	{attribute 'TcIecLibraryType'}
	{attribute 'external_name' := 'F_VN_FillContainerExp_DINT_GUID_B8D760C9_9A91_36E7_2F02_343FAF2948AF'}
	(* Partially fill the container with the specified value. Only possible for containers with basic elements. (expert function) *)
	FUNCTION F_VN_FillContainerExp_DINT : HRESULT
	VAR_INPUT
		ipContainer	:	ITcVnContainer;	(* Container with basic elements *)
		nValue	:	DINT;	(* Value to set the container elements *)
		nStartIdx	:	ULINT;	(* Start index *)
		nCount	:	ULINT;	(* Number of elements to set *)
		hrPrev	:	HRESULT;	(* HRESULT indicating the result of previous operations (If SUCCEEDED(hrPrev) equals false, no operation is executed.) *)
	END_VAR

END_FUNCTION

// Functions/Basic Container Operations/F_VN_FillContainerExp/F_VN_FillContainerExp_INT

	{attribute 'TcIecLibraryType'}
	{attribute 'external_name' := 'F_VN_FillContainerExp_INT_GUID_A3061951_E171_30F2_325A_8D22B4BE511B'}
	(* Partially fill the container with the specified value. Only possible for containers with basic elements. (expert function) *)
	FUNCTION F_VN_FillContainerExp_INT : HRESULT
	VAR_INPUT
		ipContainer	:	ITcVnContainer;	(* Container with basic elements *)
		nValue	:	INT;	(* Value to set the container elements *)
		nStartIdx	:	ULINT;	(* Start index *)
		nCount	:	ULINT;	(* Number of elements to set *)
		hrPrev	:	HRESULT;	(* HRESULT indicating the result of previous operations (If SUCCEEDED(hrPrev) equals false, no operation is executed.) *)
	END_VAR

END_FUNCTION

// Functions/Basic Container Operations/F_VN_FillContainerExp/F_VN_FillContainerExp_LREAL

	{attribute 'TcIecLibraryType'}
	{attribute 'external_name' := 'F_VN_FillContainerExp_LREAL_GUID_06A8F434_857D_380E_270C_C4307A69FA69'}
	(* Partially fill the container with the specified value. Only possible for containers with basic elements. (expert function) *)
	FUNCTION F_VN_FillContainerExp_LREAL : HRESULT
	VAR_INPUT
		ipContainer	:	ITcVnContainer;	(* Container with basic elements *)
		fValue	:	LREAL;	(* Value to set the container elements *)
		nStartIdx	:	ULINT;	(* Start index *)
		nCount	:	ULINT;	(* Number of elements to set *)
		hrPrev	:	HRESULT;	(* HRESULT indicating the result of previous operations (If SUCCEEDED(hrPrev) equals false, no operation is executed.) *)
	END_VAR

END_FUNCTION

// Functions/Basic Container Operations/F_VN_FillContainerExp/F_VN_FillContainerExp_REAL

	{attribute 'TcIecLibraryType'}
	{attribute 'external_name' := 'F_VN_FillContainerExp_REAL_GUID_48B84723_9FA9_3BC4_17C9_53CEC0ED83BA'}
	(* Partially fill the container with the specified value. Only possible for containers with basic elements. (expert function) *)
	FUNCTION F_VN_FillContainerExp_REAL : HRESULT
	VAR_INPUT
		ipContainer	:	ITcVnContainer;	(* Container with basic elements *)
		fValue	:	REAL;	(* Value to set the container elements *)
		nStartIdx	:	ULINT;	(* Start index *)
		nCount	:	ULINT;	(* Number of elements to set *)
		hrPrev	:	HRESULT;	(* HRESULT indicating the result of previous operations (If SUCCEEDED(hrPrev) equals false, no operation is executed.) *)
	END_VAR

END_FUNCTION

// Functions/Basic Container Operations/F_VN_FillContainerExp/F_VN_FillContainerExp_SINT

	{attribute 'TcIecLibraryType'}
	{attribute 'external_name' := 'F_VN_FillContainerExp_SINT_GUID_90863D28_18FF_36C8_1D3D_E4D2F13A07DE'}
	(* Partially fill the container with the specified value. Only possible for containers with basic elements. (expert function) *)
	FUNCTION F_VN_FillContainerExp_SINT : HRESULT
	VAR_INPUT
		ipContainer	:	ITcVnContainer;	(* Container with basic elements *)
		nValue	:	SINT;	(* Value to set the container elements *)
		nStartIdx	:	ULINT;	(* Start index *)
		nCount	:	ULINT;	(* Number of elements to set *)
		hrPrev	:	HRESULT;	(* HRESULT indicating the result of previous operations (If SUCCEEDED(hrPrev) equals false, no operation is executed.) *)
	END_VAR

END_FUNCTION

// Functions/Basic Container Operations/F_VN_FillContainerExp/F_VN_FillContainerExp_TcVnDMatch

	{attribute 'TcIecLibraryType'}
	{attribute 'external_name' := 'F_VN_FillContainerExp_TcVnDMatch_GUID_6EB328C8_9097_3649_0A18_3E606C0AB86C'}
	(* Partially fill the container with the specified value. Only possible for containers with basic elements. (expert function) *)
	FUNCTION F_VN_FillContainerExp_TcVnDMatch : HRESULT
	VAR_INPUT
		ipContainer	:	ITcVnContainer;	(* Container with basic elements *)
		stValue	:	REFERENCE TO TcVnDMatch;	(* Value to set the container elements *)
		nStartIdx	:	ULINT;	(* Start index *)
		nCount	:	ULINT;	(* Number of elements to set *)
		hrPrev	:	HRESULT;	(* HRESULT indicating the result of previous operations (If SUCCEEDED(hrPrev) equals false, no operation is executed.) *)
	END_VAR

END_FUNCTION

// Functions/Basic Container Operations/F_VN_FillContainerExp/F_VN_FillContainerExp_TcVnKeyPoint

	{attribute 'TcIecLibraryType'}
	{attribute 'external_name' := 'F_VN_FillContainerExp_TcVnKeyPoint_GUID_5E8CE577_86A2_3A7E_2E7B_5803657A1F81'}
	(* Partially fill the container with the specified value. Only possible for containers with basic elements. (expert function) *)
	FUNCTION F_VN_FillContainerExp_TcVnKeyPoint : HRESULT
	VAR_INPUT
		ipContainer	:	ITcVnContainer;	(* Container with basic elements *)
		stValue	:	REFERENCE TO TcVnKeyPoint;	(* Value to set the container elements *)
		nStartIdx	:	ULINT;	(* Start index *)
		nCount	:	ULINT;	(* Number of elements to set *)
		hrPrev	:	HRESULT;	(* HRESULT indicating the result of previous operations (If SUCCEEDED(hrPrev) equals false, no operation is executed.) *)
	END_VAR

END_FUNCTION

// Functions/Basic Container Operations/F_VN_FillContainerExp/F_VN_FillContainerExp_TcVnPoint2_DINT

	{attribute 'TcIecLibraryType'}
	{attribute 'external_name' := 'F_VN_FillContainerExp_TcVnPoint2_DINT_GUID_55F98272_BEB2_360C_30F1_C03770A26F61'}
	(* Partially fill the container with the specified value. Only possible for containers with basic elements. (expert function) *)
	FUNCTION F_VN_FillContainerExp_TcVnPoint2_DINT : HRESULT
	VAR_INPUT
		ipContainer	:	ITcVnContainer;	(* Container with basic elements *)
		aValue	:	REFERENCE TO TcVnPoint2_DINT;	(* Value to set the container elements *)
		nStartIdx	:	ULINT;	(* Start index *)
		nCount	:	ULINT;	(* Number of elements to set *)
		hrPrev	:	HRESULT;	(* HRESULT indicating the result of previous operations (If SUCCEEDED(hrPrev) equals false, no operation is executed.) *)
	END_VAR

END_FUNCTION

// Functions/Basic Container Operations/F_VN_FillContainerExp/F_VN_FillContainerExp_TcVnPoint2_LREAL

	{attribute 'TcIecLibraryType'}
	{attribute 'external_name' := 'F_VN_FillContainerExp_TcVnPoint2_LREAL_GUID_EFF1B11E_5960_30D8_0E25_714BE31C3872'}
	(* Partially fill the container with the specified value. Only possible for containers with basic elements. (expert function) *)
	FUNCTION F_VN_FillContainerExp_TcVnPoint2_LREAL : HRESULT
	VAR_INPUT
		ipContainer	:	ITcVnContainer;	(* Container with basic elements *)
		aValue	:	REFERENCE TO TcVnPoint2_LREAL;	(* Value to set the container elements *)
		nStartIdx	:	ULINT;	(* Start index *)
		nCount	:	ULINT;	(* Number of elements to set *)
		hrPrev	:	HRESULT;	(* HRESULT indicating the result of previous operations (If SUCCEEDED(hrPrev) equals false, no operation is executed.) *)
	END_VAR

END_FUNCTION

// Functions/Basic Container Operations/F_VN_FillContainerExp/F_VN_FillContainerExp_TcVnPoint2_REAL

	{attribute 'TcIecLibraryType'}
	{attribute 'external_name' := 'F_VN_FillContainerExp_TcVnPoint2_REAL_GUID_D2951393_83B9_352D_040D_B4C5DB5D1089'}
	(* Partially fill the container with the specified value. Only possible for containers with basic elements. (expert function) *)
	FUNCTION F_VN_FillContainerExp_TcVnPoint2_REAL : HRESULT
	VAR_INPUT
		ipContainer	:	ITcVnContainer;	(* Container with basic elements *)
		aValue	:	REFERENCE TO TcVnPoint2_REAL;	(* Value to set the container elements *)
		nStartIdx	:	ULINT;	(* Start index *)
		nCount	:	ULINT;	(* Number of elements to set *)
		hrPrev	:	HRESULT;	(* HRESULT indicating the result of previous operations (If SUCCEEDED(hrPrev) equals false, no operation is executed.) *)
	END_VAR

END_FUNCTION

// Functions/Basic Container Operations/F_VN_FillContainerExp/F_VN_FillContainerExp_TcVnPoint3_LREAL

	{attribute 'TcIecLibraryType'}
	{attribute 'external_name' := 'F_VN_FillContainerExp_TcVnPoint3_LREAL_GUID_B768B07E_F5CA_3309_10EA_C90BF763008C'}
	(* Partially fill the container with the specified value. Only possible for containers with basic elements. (expert function) *)
	FUNCTION F_VN_FillContainerExp_TcVnPoint3_LREAL : HRESULT
	VAR_INPUT
		ipContainer	:	ITcVnContainer;	(* Container with basic elements *)
		aValue	:	REFERENCE TO TcVnPoint3_LREAL;	(* Value to set the container elements *)
		nStartIdx	:	ULINT;	(* Start index *)
		nCount	:	ULINT;	(* Number of elements to set *)
		hrPrev	:	HRESULT;	(* HRESULT indicating the result of previous operations (If SUCCEEDED(hrPrev) equals false, no operation is executed.) *)
	END_VAR

END_FUNCTION

// Functions/Basic Container Operations/F_VN_FillContainerExp/F_VN_FillContainerExp_TcVnPoint3_REAL

	{attribute 'TcIecLibraryType'}
	{attribute 'external_name' := 'F_VN_FillContainerExp_TcVnPoint3_REAL_GUID_6AD4CB96_3415_3337_191D_E41E5C35A24A'}
	(* Partially fill the container with the specified value. Only possible for containers with basic elements. (expert function) *)
	FUNCTION F_VN_FillContainerExp_TcVnPoint3_REAL : HRESULT
	VAR_INPUT
		ipContainer	:	ITcVnContainer;	(* Container with basic elements *)
		aValue	:	REFERENCE TO TcVnPoint3_REAL;	(* Value to set the container elements *)
		nStartIdx	:	ULINT;	(* Start index *)
		nCount	:	ULINT;	(* Number of elements to set *)
		hrPrev	:	HRESULT;	(* HRESULT indicating the result of previous operations (If SUCCEEDED(hrPrev) equals false, no operation is executed.) *)
	END_VAR

END_FUNCTION

// Functions/Basic Container Operations/F_VN_FillContainerExp/F_VN_FillContainerExp_TcVnRectangle_DINT

	{attribute 'TcIecLibraryType'}
	{attribute 'external_name' := 'F_VN_FillContainerExp_TcVnRectangle_DINT_GUID_8BBC2A7F_64C7_3525_1E97_8C907D649B01'}
	(* Partially fill the container with the specified value. Only possible for containers with basic elements. (expert function) *)
	FUNCTION F_VN_FillContainerExp_TcVnRectangle_DINT : HRESULT
	VAR_INPUT
		ipContainer	:	ITcVnContainer;	(* Container with basic elements *)
		stValue	:	REFERENCE TO TcVnRectangle_DINT;	(* Value to set the container elements *)
		nStartIdx	:	ULINT;	(* Start index *)
		nCount	:	ULINT;	(* Number of elements to set *)
		hrPrev	:	HRESULT;	(* HRESULT indicating the result of previous operations (If SUCCEEDED(hrPrev) equals false, no operation is executed.) *)
	END_VAR

END_FUNCTION

// Functions/Basic Container Operations/F_VN_FillContainerExp/F_VN_FillContainerExp_TcVnVector2_DINT

	{attribute 'TcIecLibraryType'}
	{attribute 'external_name' := 'F_VN_FillContainerExp_TcVnVector2_DINT_GUID_D52E6A94_DE58_3796_0B33_2DB8E1E8C278'}
	(* Partially fill the container with the specified value. Only possible for containers with basic elements. (expert function) *)
	FUNCTION F_VN_FillContainerExp_TcVnVector2_DINT : HRESULT
	VAR_INPUT
		ipContainer	:	ITcVnContainer;	(* Container with basic elements *)
		aValue	:	REFERENCE TO TcVnVector2_DINT;	(* Value to set the container elements *)
		nStartIdx	:	ULINT;	(* Start index *)
		nCount	:	ULINT;	(* Number of elements to set *)
		hrPrev	:	HRESULT;	(* HRESULT indicating the result of previous operations (If SUCCEEDED(hrPrev) equals false, no operation is executed.) *)
	END_VAR

END_FUNCTION

// Functions/Basic Container Operations/F_VN_FillContainerExp/F_VN_FillContainerExp_TcVnVector2_INT

	{attribute 'TcIecLibraryType'}
	{attribute 'external_name' := 'F_VN_FillContainerExp_TcVnVector2_INT_GUID_F0AB717A_FE22_3EAE_3CD4_F3F145D668E6'}
	(* Partially fill the container with the specified value. Only possible for containers with basic elements. (expert function) *)
	FUNCTION F_VN_FillContainerExp_TcVnVector2_INT : HRESULT
	VAR_INPUT
		ipContainer	:	ITcVnContainer;	(* Container with basic elements *)
		aValue	:	REFERENCE TO TcVnVector2_INT;	(* Value to set the container elements *)
		nStartIdx	:	ULINT;	(* Start index *)
		nCount	:	ULINT;	(* Number of elements to set *)
		hrPrev	:	HRESULT;	(* HRESULT indicating the result of previous operations (If SUCCEEDED(hrPrev) equals false, no operation is executed.) *)
	END_VAR

END_FUNCTION

// Functions/Basic Container Operations/F_VN_FillContainerExp/F_VN_FillContainerExp_TcVnVector2_REAL

	{attribute 'TcIecLibraryType'}
	{attribute 'external_name' := 'F_VN_FillContainerExp_TcVnVector2_REAL_GUID_79D3ED73_D9A1_3766_3CCC_01A7C4952E54'}
	(* Partially fill the container with the specified value. Only possible for containers with basic elements. (expert function) *)
	FUNCTION F_VN_FillContainerExp_TcVnVector2_REAL : HRESULT
	VAR_INPUT
		ipContainer	:	ITcVnContainer;	(* Container with basic elements *)
		aValue	:	REFERENCE TO TcVnVector2_REAL;	(* Value to set the container elements *)
		nStartIdx	:	ULINT;	(* Start index *)
		nCount	:	ULINT;	(* Number of elements to set *)
		hrPrev	:	HRESULT;	(* HRESULT indicating the result of previous operations (If SUCCEEDED(hrPrev) equals false, no operation is executed.) *)
	END_VAR

END_FUNCTION

// Functions/Basic Container Operations/F_VN_FillContainerExp/F_VN_FillContainerExp_TcVnVector2_SINT

	{attribute 'TcIecLibraryType'}
	{attribute 'external_name' := 'F_VN_FillContainerExp_TcVnVector2_SINT_GUID_5A606FB7_F136_3298_1B9E_CE3509B64A28'}
	(* Partially fill the container with the specified value. Only possible for containers with basic elements. (expert function) *)
	FUNCTION F_VN_FillContainerExp_TcVnVector2_SINT : HRESULT
	VAR_INPUT
		ipContainer	:	ITcVnContainer;	(* Container with basic elements *)
		aValue	:	REFERENCE TO TcVnVector2_SINT;	(* Value to set the container elements *)
		nStartIdx	:	ULINT;	(* Start index *)
		nCount	:	ULINT;	(* Number of elements to set *)
		hrPrev	:	HRESULT;	(* HRESULT indicating the result of previous operations (If SUCCEEDED(hrPrev) equals false, no operation is executed.) *)
	END_VAR

END_FUNCTION

// Functions/Basic Container Operations/F_VN_FillContainerExp/F_VN_FillContainerExp_TcVnVector2_UINT

	{attribute 'TcIecLibraryType'}
	{attribute 'external_name' := 'F_VN_FillContainerExp_TcVnVector2_UINT_GUID_28D7E1DD_8953_3773_2801_6C09CC21C0E8'}
	(* Partially fill the container with the specified value. Only possible for containers with basic elements. (expert function) *)
	FUNCTION F_VN_FillContainerExp_TcVnVector2_UINT : HRESULT
	VAR_INPUT
		ipContainer	:	ITcVnContainer;	(* Container with basic elements *)
		aValue	:	REFERENCE TO TcVnVector2_UINT;	(* Value to set the container elements *)
		nStartIdx	:	ULINT;	(* Start index *)
		nCount	:	ULINT;	(* Number of elements to set *)
		hrPrev	:	HRESULT;	(* HRESULT indicating the result of previous operations (If SUCCEEDED(hrPrev) equals false, no operation is executed.) *)
	END_VAR

END_FUNCTION

// Functions/Basic Container Operations/F_VN_FillContainerExp/F_VN_FillContainerExp_TcVnVector2_USINT

	{attribute 'TcIecLibraryType'}
	{attribute 'external_name' := 'F_VN_FillContainerExp_TcVnVector2_USINT_GUID_CADE4DE9_E251_30AB_3613_56AF17179610'}
	(* Partially fill the container with the specified value. Only possible for containers with basic elements. (expert function) *)
	FUNCTION F_VN_FillContainerExp_TcVnVector2_USINT : HRESULT
	VAR_INPUT
		ipContainer	:	ITcVnContainer;	(* Container with basic elements *)
		aValue	:	REFERENCE TO TcVnVector2_USINT;	(* Value to set the container elements *)
		nStartIdx	:	ULINT;	(* Start index *)
		nCount	:	ULINT;	(* Number of elements to set *)
		hrPrev	:	HRESULT;	(* HRESULT indicating the result of previous operations (If SUCCEEDED(hrPrev) equals false, no operation is executed.) *)
	END_VAR

END_FUNCTION

// Functions/Basic Container Operations/F_VN_FillContainerExp/F_VN_FillContainerExp_TcVnVector3_INT

	{attribute 'TcIecLibraryType'}
	{attribute 'external_name' := 'F_VN_FillContainerExp_TcVnVector3_INT_GUID_8872692A_8B44_3770_16B3_D8C1614F2555'}
	(* Partially fill the container with the specified value. Only possible for containers with basic elements. (expert function) *)
	FUNCTION F_VN_FillContainerExp_TcVnVector3_INT : HRESULT
	VAR_INPUT
		ipContainer	:	ITcVnContainer;	(* Container with basic elements *)
		aValue	:	REFERENCE TO TcVnVector3_INT;	(* Value to set the container elements *)
		nStartIdx	:	ULINT;	(* Start index *)
		nCount	:	ULINT;	(* Number of elements to set *)
		hrPrev	:	HRESULT;	(* HRESULT indicating the result of previous operations (If SUCCEEDED(hrPrev) equals false, no operation is executed.) *)
	END_VAR

END_FUNCTION

// Functions/Basic Container Operations/F_VN_FillContainerExp/F_VN_FillContainerExp_TcVnVector3_REAL

	{attribute 'TcIecLibraryType'}
	{attribute 'external_name' := 'F_VN_FillContainerExp_TcVnVector3_REAL_GUID_F71E09F4_5F32_3920_383B_6FAF0F1CEF00'}
	(* Partially fill the container with the specified value. Only possible for containers with basic elements. (expert function) *)
	FUNCTION F_VN_FillContainerExp_TcVnVector3_REAL : HRESULT
	VAR_INPUT
		ipContainer	:	ITcVnContainer;	(* Container with basic elements *)
		aValue	:	REFERENCE TO TcVnVector3_REAL;	(* Value to set the container elements *)
		nStartIdx	:	ULINT;	(* Start index *)
		nCount	:	ULINT;	(* Number of elements to set *)
		hrPrev	:	HRESULT;	(* HRESULT indicating the result of previous operations (If SUCCEEDED(hrPrev) equals false, no operation is executed.) *)
	END_VAR

END_FUNCTION

// Functions/Basic Container Operations/F_VN_FillContainerExp/F_VN_FillContainerExp_TcVnVector3_SINT

	{attribute 'TcIecLibraryType'}
	{attribute 'external_name' := 'F_VN_FillContainerExp_TcVnVector3_SINT_GUID_C767BF5E_81CB_35B7_2F21_D703B6074D66'}
	(* Partially fill the container with the specified value. Only possible for containers with basic elements. (expert function) *)
	FUNCTION F_VN_FillContainerExp_TcVnVector3_SINT : HRESULT
	VAR_INPUT
		ipContainer	:	ITcVnContainer;	(* Container with basic elements *)
		aValue	:	REFERENCE TO TcVnVector3_SINT;	(* Value to set the container elements *)
		nStartIdx	:	ULINT;	(* Start index *)
		nCount	:	ULINT;	(* Number of elements to set *)
		hrPrev	:	HRESULT;	(* HRESULT indicating the result of previous operations (If SUCCEEDED(hrPrev) equals false, no operation is executed.) *)
	END_VAR

END_FUNCTION

// Functions/Basic Container Operations/F_VN_FillContainerExp/F_VN_FillContainerExp_TcVnVector3_UINT

	{attribute 'TcIecLibraryType'}
	{attribute 'external_name' := 'F_VN_FillContainerExp_TcVnVector3_UINT_GUID_A232C566_3D1F_3878_20BE_EC4C243376B7'}
	(* Partially fill the container with the specified value. Only possible for containers with basic elements. (expert function) *)
	FUNCTION F_VN_FillContainerExp_TcVnVector3_UINT : HRESULT
	VAR_INPUT
		ipContainer	:	ITcVnContainer;	(* Container with basic elements *)
		aValue	:	REFERENCE TO TcVnVector3_UINT;	(* Value to set the container elements *)
		nStartIdx	:	ULINT;	(* Start index *)
		nCount	:	ULINT;	(* Number of elements to set *)
		hrPrev	:	HRESULT;	(* HRESULT indicating the result of previous operations (If SUCCEEDED(hrPrev) equals false, no operation is executed.) *)
	END_VAR

END_FUNCTION

// Functions/Basic Container Operations/F_VN_FillContainerExp/F_VN_FillContainerExp_TcVnVector3_USINT

	{attribute 'TcIecLibraryType'}
	{attribute 'external_name' := 'F_VN_FillContainerExp_TcVnVector3_USINT_GUID_AF77E3C4_6637_32BB_0907_3628D17ABB88'}
	(* Partially fill the container with the specified value. Only possible for containers with basic elements. (expert function) *)
	FUNCTION F_VN_FillContainerExp_TcVnVector3_USINT : HRESULT
	VAR_INPUT
		ipContainer	:	ITcVnContainer;	(* Container with basic elements *)
		aValue	:	REFERENCE TO TcVnVector3_USINT;	(* Value to set the container elements *)
		nStartIdx	:	ULINT;	(* Start index *)
		nCount	:	ULINT;	(* Number of elements to set *)
		hrPrev	:	HRESULT;	(* HRESULT indicating the result of previous operations (If SUCCEEDED(hrPrev) equals false, no operation is executed.) *)
	END_VAR

END_FUNCTION

// Functions/Basic Container Operations/F_VN_FillContainerExp/F_VN_FillContainerExp_TcVnVector4_DINT

	{attribute 'TcIecLibraryType'}
	{attribute 'external_name' := 'F_VN_FillContainerExp_TcVnVector4_DINT_GUID_D0B471BF_D0B3_3250_3545_D00683C80B71'}
	(* Partially fill the container with the specified value. Only possible for containers with basic elements. (expert function) *)
	FUNCTION F_VN_FillContainerExp_TcVnVector4_DINT : HRESULT
	VAR_INPUT
		ipContainer	:	ITcVnContainer;	(* Container with basic elements *)
		aValue	:	REFERENCE TO TcVnVector4_DINT;	(* Value to set the container elements *)
		nStartIdx	:	ULINT;	(* Start index *)
		nCount	:	ULINT;	(* Number of elements to set *)
		hrPrev	:	HRESULT;	(* HRESULT indicating the result of previous operations (If SUCCEEDED(hrPrev) equals false, no operation is executed.) *)
	END_VAR

END_FUNCTION

// Functions/Basic Container Operations/F_VN_FillContainerExp/F_VN_FillContainerExp_TcVnVector4_INT

	{attribute 'TcIecLibraryType'}
	{attribute 'external_name' := 'F_VN_FillContainerExp_TcVnVector4_INT_GUID_FE07D4F2_2BAB_357F_1E6D_1BC89319641C'}
	(* Partially fill the container with the specified value. Only possible for containers with basic elements. (expert function) *)
	FUNCTION F_VN_FillContainerExp_TcVnVector4_INT : HRESULT
	VAR_INPUT
		ipContainer	:	ITcVnContainer;	(* Container with basic elements *)
		aValue	:	REFERENCE TO TcVnVector4_INT;	(* Value to set the container elements *)
		nStartIdx	:	ULINT;	(* Start index *)
		nCount	:	ULINT;	(* Number of elements to set *)
		hrPrev	:	HRESULT;	(* HRESULT indicating the result of previous operations (If SUCCEEDED(hrPrev) equals false, no operation is executed.) *)
	END_VAR

END_FUNCTION

// Functions/Basic Container Operations/F_VN_FillContainerExp/F_VN_FillContainerExp_TcVnVector4_LREAL

	{attribute 'TcIecLibraryType'}
	{attribute 'external_name' := 'F_VN_FillContainerExp_TcVnVector4_LREAL_GUID_DE917028_E855_3AAC_2584_39BC076C3EA3'}
	(* Partially fill the container with the specified value. Only possible for containers with basic elements. (expert function) *)
	FUNCTION F_VN_FillContainerExp_TcVnVector4_LREAL : HRESULT
	VAR_INPUT
		ipContainer	:	ITcVnContainer;	(* Container with basic elements *)
		aValue	:	REFERENCE TO TcVnVector4_LREAL;	(* Value to set the container elements *)
		nStartIdx	:	ULINT;	(* Start index *)
		nCount	:	ULINT;	(* Number of elements to set *)
		hrPrev	:	HRESULT;	(* HRESULT indicating the result of previous operations (If SUCCEEDED(hrPrev) equals false, no operation is executed.) *)
	END_VAR

END_FUNCTION

// Functions/Basic Container Operations/F_VN_FillContainerExp/F_VN_FillContainerExp_TcVnVector4_SINT

	{attribute 'TcIecLibraryType'}
	{attribute 'external_name' := 'F_VN_FillContainerExp_TcVnVector4_SINT_GUID_36AF45DF_9EEE_3748_11FA_C0473793B250'}
	(* Partially fill the container with the specified value. Only possible for containers with basic elements. (expert function) *)
	FUNCTION F_VN_FillContainerExp_TcVnVector4_SINT : HRESULT
	VAR_INPUT
		ipContainer	:	ITcVnContainer;	(* Container with basic elements *)
		aValue	:	REFERENCE TO TcVnVector4_SINT;	(* Value to set the container elements *)
		nStartIdx	:	ULINT;	(* Start index *)
		nCount	:	ULINT;	(* Number of elements to set *)
		hrPrev	:	HRESULT;	(* HRESULT indicating the result of previous operations (If SUCCEEDED(hrPrev) equals false, no operation is executed.) *)
	END_VAR

END_FUNCTION

// Functions/Basic Container Operations/F_VN_FillContainerExp/F_VN_FillContainerExp_TcVnVector4_UINT

	{attribute 'TcIecLibraryType'}
	{attribute 'external_name' := 'F_VN_FillContainerExp_TcVnVector4_UINT_GUID_6F025B14_1449_32FD_3652_7705ACD933FC'}
	(* Partially fill the container with the specified value. Only possible for containers with basic elements. (expert function) *)
	FUNCTION F_VN_FillContainerExp_TcVnVector4_UINT : HRESULT
	VAR_INPUT
		ipContainer	:	ITcVnContainer;	(* Container with basic elements *)
		aValue	:	REFERENCE TO TcVnVector4_UINT;	(* Value to set the container elements *)
		nStartIdx	:	ULINT;	(* Start index *)
		nCount	:	ULINT;	(* Number of elements to set *)
		hrPrev	:	HRESULT;	(* HRESULT indicating the result of previous operations (If SUCCEEDED(hrPrev) equals false, no operation is executed.) *)
	END_VAR

END_FUNCTION

// Functions/Basic Container Operations/F_VN_FillContainerExp/F_VN_FillContainerExp_TcVnVector4_USINT

	{attribute 'TcIecLibraryType'}
	{attribute 'external_name' := 'F_VN_FillContainerExp_TcVnVector4_USINT_GUID_88F61DD9_1D3A_3F92_2879_A4E50CB6EE10'}
	(* Partially fill the container with the specified value. Only possible for containers with basic elements. (expert function) *)
	FUNCTION F_VN_FillContainerExp_TcVnVector4_USINT : HRESULT
	VAR_INPUT
		ipContainer	:	ITcVnContainer;	(* Container with basic elements *)
		aValue	:	REFERENCE TO TcVnVector4_USINT;	(* Value to set the container elements *)
		nStartIdx	:	ULINT;	(* Start index *)
		nCount	:	ULINT;	(* Number of elements to set *)
		hrPrev	:	HRESULT;	(* HRESULT indicating the result of previous operations (If SUCCEEDED(hrPrev) equals false, no operation is executed.) *)
	END_VAR

END_FUNCTION

// Functions/Basic Container Operations/F_VN_FillContainerExp/F_VN_FillContainerExp_UDINT

	{attribute 'TcIecLibraryType'}
	{attribute 'external_name' := 'F_VN_FillContainerExp_UDINT_GUID_C1899B3C_8E1E_3688_3F00_9FEF7C4BAF80'}
	(* Partially fill the container with the specified value. Only possible for containers with basic elements. (expert function) *)
	FUNCTION F_VN_FillContainerExp_UDINT : HRESULT
	VAR_INPUT
		ipContainer	:	ITcVnContainer;	(* Container with basic elements *)
		nValue	:	UDINT;	(* Value to set the container elements *)
		nStartIdx	:	ULINT;	(* Start index *)
		nCount	:	ULINT;	(* Number of elements to set *)
		hrPrev	:	HRESULT;	(* HRESULT indicating the result of previous operations (If SUCCEEDED(hrPrev) equals false, no operation is executed.) *)
	END_VAR

END_FUNCTION

// Functions/Basic Container Operations/F_VN_FillContainerExp/F_VN_FillContainerExp_UINT

	{attribute 'TcIecLibraryType'}
	{attribute 'external_name' := 'F_VN_FillContainerExp_UINT_GUID_4625D03C_9DE0_3ACB_0D71_512E8D91ACEF'}
	(* Partially fill the container with the specified value. Only possible for containers with basic elements. (expert function) *)
	FUNCTION F_VN_FillContainerExp_UINT : HRESULT
	VAR_INPUT
		ipContainer	:	ITcVnContainer;	(* Container with basic elements *)
		nValue	:	UINT;	(* Value to set the container elements *)
		nStartIdx	:	ULINT;	(* Start index *)
		nCount	:	ULINT;	(* Number of elements to set *)
		hrPrev	:	HRESULT;	(* HRESULT indicating the result of previous operations (If SUCCEEDED(hrPrev) equals false, no operation is executed.) *)
	END_VAR

END_FUNCTION

// Functions/Basic Container Operations/F_VN_FillContainerExp/F_VN_FillContainerExp_ULINT

	{attribute 'TcIecLibraryType'}
	{attribute 'external_name' := 'F_VN_FillContainerExp_ULINT_GUID_E1571213_CE5E_37DB_3EDB_D35295DEA11A'}
	(* Partially fill the container with the specified value. Only possible for containers with basic elements. (expert function) *)
	FUNCTION F_VN_FillContainerExp_ULINT : HRESULT
	VAR_INPUT
		ipContainer	:	ITcVnContainer;	(* Container with basic elements *)
		nValue	:	ULINT;	(* Value to set the container elements *)
		nStartIdx	:	ULINT;	(* Start index *)
		nCount	:	ULINT;	(* Number of elements to set *)
		hrPrev	:	HRESULT;	(* HRESULT indicating the result of previous operations (If SUCCEEDED(hrPrev) equals false, no operation is executed.) *)
	END_VAR

END_FUNCTION

// Functions/Basic Container Operations/F_VN_FillContainerExp/F_VN_FillContainerExp_USINT

	{attribute 'TcIecLibraryType'}
	{attribute 'external_name' := 'F_VN_FillContainerExp_USINT_GUID_5EEE187D_276D_381A_26F0_6B86E27B5CD0'}
	(* Partially fill the container with the specified value. Only possible for containers with basic elements. (expert function) *)
	FUNCTION F_VN_FillContainerExp_USINT : HRESULT
	VAR_INPUT
		ipContainer	:	ITcVnContainer;	(* Container with basic elements *)
		nValue	:	USINT;	(* Value to set the container elements *)
		nStartIdx	:	ULINT;	(* Start index *)
		nCount	:	ULINT;	(* Number of elements to set *)
		hrPrev	:	HRESULT;	(* HRESULT indicating the result of previous operations (If SUCCEEDED(hrPrev) equals false, no operation is executed.) *)
	END_VAR

END_FUNCTION

// Functions/Basic Container Operations/F_VN_GetAt/F_VN_GetAt_ITcVnContainer

	{attribute 'TcIecLibraryType'}
	{attribute 'external_name' := 'F_VN_GetAt_ITcVnContainer_GUID_045FB529_DC44_35D8_25B4_376FBA31652E'}
	(* Gets the ITcVnContainer element at the specified index of the source container. (Alternatively use interface method .GetAt.) *)
	FUNCTION F_VN_GetAt_ITcVnContainer : HRESULT
	VAR_INPUT
		ipSrcContainer	:	ITcVnContainer;	(* Container with ITcVnContainer elements *)
		ipDestContainer	:	REFERENCE TO ITcVnContainer;	(* Returns the container at the specified index *)
		nIndex	:	ULINT;	(* Index of the requested element *)
		hrPrev	:	HRESULT;	(* HRESULT indicating the result of previous operations (If SUCCEEDED(hrPrev) equals false, no operation is executed.) *)
	END_VAR

END_FUNCTION

// Functions/Basic Container Operations/F_VN_GetAt/F_VN_GetAt_DINT

	{attribute 'TcIecLibraryType'}
	{attribute 'external_name' := 'F_VN_GetAt_DINT_GUID_D3F93AB3_14EE_32CD_0E8F_11068B05A3A3'}
	(* Gets the DINT element at the specified index of the container. *)
	FUNCTION F_VN_GetAt_DINT : HRESULT
	VAR_INPUT
		ipContainer	:	ITcVnContainer;	(* Container with DINT elements *)
		nElement	:	REFERENCE TO DINT;	(* Returns the element at the specified index *)
		nIndex	:	ULINT;	(* Index of the requested element *)
		hrPrev	:	HRESULT;	(* HRESULT indicating the result of previous operations (If SUCCEEDED(hrPrev) equals false, no operation is executed.) *)
	END_VAR

END_FUNCTION

// Functions/Basic Container Operations/F_VN_GetAt/F_VN_GetAt_INT

	{attribute 'TcIecLibraryType'}
	{attribute 'external_name' := 'F_VN_GetAt_INT_GUID_9B8341DD_2E11_3864_2634_BD22319F2AE6'}
	(* Gets the INT element at the specified index of the container. *)
	FUNCTION F_VN_GetAt_INT : HRESULT
	VAR_INPUT
		ipContainer	:	ITcVnContainer;	(* Container with INT elements *)
		nElement	:	REFERENCE TO INT;	(* Returns the element at the specified index *)
		nIndex	:	ULINT;	(* Index of the requested element *)
		hrPrev	:	HRESULT;	(* HRESULT indicating the result of previous operations (If SUCCEEDED(hrPrev) equals false, no operation is executed.) *)
	END_VAR

END_FUNCTION

// Functions/Basic Container Operations/F_VN_GetAt/F_VN_GetAt_LREAL

	{attribute 'TcIecLibraryType'}
	{attribute 'external_name' := 'F_VN_GetAt_LREAL_GUID_DC876A81_A8A4_3799_1F06_D74BAE2F1D06'}
	(* Gets the LREAL element at the specified index of the container. *)
	FUNCTION F_VN_GetAt_LREAL : HRESULT
	VAR_INPUT
		ipContainer	:	ITcVnContainer;	(* Container with LREAL elements *)
		fElement	:	REFERENCE TO LREAL;	(* Returns the element at the specified index *)
		nIndex	:	ULINT;	(* Index of the requested element *)
		hrPrev	:	HRESULT;	(* HRESULT indicating the result of previous operations (If SUCCEEDED(hrPrev) equals false, no operation is executed.) *)
	END_VAR

END_FUNCTION

// Functions/Basic Container Operations/F_VN_GetAt/F_VN_GetAt_REAL

	{attribute 'TcIecLibraryType'}
	{attribute 'external_name' := 'F_VN_GetAt_REAL_GUID_1E16943C_FBCF_3296_0945_06B3CBBED3E4'}
	(* Gets the REAL element at the specified index of the container. *)
	FUNCTION F_VN_GetAt_REAL : HRESULT
	VAR_INPUT
		ipContainer	:	ITcVnContainer;	(* Container with REAL elements *)
		fElement	:	REFERENCE TO REAL;	(* Returns the element at the specified index *)
		nIndex	:	ULINT;	(* Index of the requested element *)
		hrPrev	:	HRESULT;	(* HRESULT indicating the result of previous operations (If SUCCEEDED(hrPrev) equals false, no operation is executed.) *)
	END_VAR

END_FUNCTION

// Functions/Basic Container Operations/F_VN_GetAt/F_VN_GetAt_SINT

	{attribute 'TcIecLibraryType'}
	{attribute 'external_name' := 'F_VN_GetAt_SINT_GUID_881646F0_463E_317B_2E29_F707EE20003C'}
	(* Gets the SINT element at the specified index of the container. *)
	FUNCTION F_VN_GetAt_SINT : HRESULT
	VAR_INPUT
		ipContainer	:	ITcVnContainer;	(* Container with SINT elements *)
		nElement	:	REFERENCE TO SINT;	(* Returns the element at the specified index *)
		nIndex	:	ULINT;	(* Index of the requested element *)
		hrPrev	:	HRESULT;	(* HRESULT indicating the result of previous operations (If SUCCEEDED(hrPrev) equals false, no operation is executed.) *)
	END_VAR

END_FUNCTION

// Functions/Basic Container Operations/F_VN_GetAt/F_VN_GetAt_TcVnDMatch

	{attribute 'TcIecLibraryType'}
	{attribute 'external_name' := 'F_VN_GetAt_TcVnDMatch_GUID_3207E963_392F_3409_08E6_68F01287B943'}
	(* Gets the TcVnDMatch element at the specified index of the container. *)
	FUNCTION F_VN_GetAt_TcVnDMatch : HRESULT
	VAR_INPUT
		ipContainer	:	ITcVnContainer;	(* Container with TcVnDMatch elements *)
		stElement	:	REFERENCE TO TcVnDMatch;	(* Returns the element at the specified index *)
		nIndex	:	ULINT;	(* Index of the requested element *)
		hrPrev	:	HRESULT;	(* HRESULT indicating the result of previous operations (If SUCCEEDED(hrPrev) equals false, no operation is executed.) *)
	END_VAR

END_FUNCTION

// Functions/Basic Container Operations/F_VN_GetAt/F_VN_GetAt_TcVnKeyPoint

	{attribute 'TcIecLibraryType'}
	{attribute 'external_name' := 'F_VN_GetAt_TcVnKeyPoint_GUID_2D05125E_4551_301B_1496_C775451626E2'}
	(* Gets the TcVnKeyPoint element at the specified index of the container. *)
	FUNCTION F_VN_GetAt_TcVnKeyPoint : HRESULT
	VAR_INPUT
		ipContainer	:	ITcVnContainer;	(* Container with TcVnKeyPoint elements *)
		stElement	:	REFERENCE TO TcVnKeyPoint;	(* Returns the element at the specified index *)
		nIndex	:	ULINT;	(* Index of the requested element *)
		hrPrev	:	HRESULT;	(* HRESULT indicating the result of previous operations (If SUCCEEDED(hrPrev) equals false, no operation is executed.) *)
	END_VAR

END_FUNCTION

// Functions/Basic Container Operations/F_VN_GetAt/F_VN_GetAt_TcVnPoint2_DINT

	{attribute 'TcIecLibraryType'}
	{attribute 'external_name' := 'F_VN_GetAt_TcVnPoint2_DINT_GUID_E33E2091_0EF8_3437_0DF4_98D7E3EF7746'}
	(* Gets the TcVnPoint2_DINT element at the specified index of the container. *)
	FUNCTION F_VN_GetAt_TcVnPoint2_DINT : HRESULT
	VAR_INPUT
		ipContainer	:	ITcVnContainer;	(* Container with TcVnPoint2_DINT elements *)
		aElement	:	REFERENCE TO TcVnPoint2_DINT;	(* Returns the element at the specified index *)
		nIndex	:	ULINT;	(* Index of the requested element *)
		hrPrev	:	HRESULT;	(* HRESULT indicating the result of previous operations (If SUCCEEDED(hrPrev) equals false, no operation is executed.) *)
	END_VAR

END_FUNCTION

// Functions/Basic Container Operations/F_VN_GetAt/F_VN_GetAt_TcVnPoint2_LREAL

	{attribute 'TcIecLibraryType'}
	{attribute 'external_name' := 'F_VN_GetAt_TcVnPoint2_LREAL_GUID_9EEB5F99_0D0C_312C_2F99_C7BA67AF2141'}
	(* Gets the TcVnPoint2_LREAL element at the specified index of the container. *)
	FUNCTION F_VN_GetAt_TcVnPoint2_LREAL : HRESULT
	VAR_INPUT
		ipContainer	:	ITcVnContainer;	(* Container with TcVnPoint2_LREAL elements *)
		aElement	:	REFERENCE TO TcVnPoint2_LREAL;	(* Returns the element at the specified index *)
		nIndex	:	ULINT;	(* Index of the requested element *)
		hrPrev	:	HRESULT;	(* HRESULT indicating the result of previous operations (If SUCCEEDED(hrPrev) equals false, no operation is executed.) *)
	END_VAR

END_FUNCTION

// Functions/Basic Container Operations/F_VN_GetAt/F_VN_GetAt_TcVnPoint2_REAL

	{attribute 'TcIecLibraryType'}
	{attribute 'external_name' := 'F_VN_GetAt_TcVnPoint2_REAL_GUID_371EAF1D_26B5_3B9D_372A_6247762CF125'}
	(* Gets the TcVnPoint2_REAL element at the specified index of the container. *)
	FUNCTION F_VN_GetAt_TcVnPoint2_REAL : HRESULT
	VAR_INPUT
		ipContainer	:	ITcVnContainer;	(* Container with TcVnPoint2_REAL elements *)
		aElement	:	REFERENCE TO TcVnPoint2_REAL;	(* Returns the element at the specified index *)
		nIndex	:	ULINT;	(* Index of the requested element *)
		hrPrev	:	HRESULT;	(* HRESULT indicating the result of previous operations (If SUCCEEDED(hrPrev) equals false, no operation is executed.) *)
	END_VAR

END_FUNCTION

// Functions/Basic Container Operations/F_VN_GetAt/F_VN_GetAt_TcVnPoint3_LREAL

	{attribute 'TcIecLibraryType'}
	{attribute 'external_name' := 'F_VN_GetAt_TcVnPoint3_LREAL_GUID_90390C07_74BB_3F31_196C_51E52FA0FEDF'}
	(* Gets the TcVnPoint3_LREAL element at the specified index of the container. *)
	FUNCTION F_VN_GetAt_TcVnPoint3_LREAL : HRESULT
	VAR_INPUT
		ipContainer	:	ITcVnContainer;	(* Container with TcVnPoint3_LREAL elements *)
		aElement	:	REFERENCE TO TcVnPoint3_LREAL;	(* Returns the element at the specified index *)
		nIndex	:	ULINT;	(* Index of the requested element *)
		hrPrev	:	HRESULT;	(* HRESULT indicating the result of previous operations (If SUCCEEDED(hrPrev) equals false, no operation is executed.) *)
	END_VAR

END_FUNCTION

// Functions/Basic Container Operations/F_VN_GetAt/F_VN_GetAt_TcVnPoint3_REAL

	{attribute 'TcIecLibraryType'}
	{attribute 'external_name' := 'F_VN_GetAt_TcVnPoint3_REAL_GUID_0A5DCE69_37A2_35F9_0DF3_FEC0A8403AF7'}
	(* Gets the TcVnPoint3_REAL element at the specified index of the container. *)
	FUNCTION F_VN_GetAt_TcVnPoint3_REAL : HRESULT
	VAR_INPUT
		ipContainer	:	ITcVnContainer;	(* Container with TcVnPoint3_REAL elements *)
		aElement	:	REFERENCE TO TcVnPoint3_REAL;	(* Returns the element at the specified index *)
		nIndex	:	ULINT;	(* Index of the requested element *)
		hrPrev	:	HRESULT;	(* HRESULT indicating the result of previous operations (If SUCCEEDED(hrPrev) equals false, no operation is executed.) *)
	END_VAR

END_FUNCTION

// Functions/Basic Container Operations/F_VN_GetAt/F_VN_GetAt_TcVnRectangle_DINT

	{attribute 'TcIecLibraryType'}
	{attribute 'external_name' := 'F_VN_GetAt_TcVnRectangle_DINT_GUID_75B34143_A1C0_32FF_0BAA_7C7E335D62E6'}
	(* Gets the TcVnRectangle_DINT element at the specified index of the container. *)
	FUNCTION F_VN_GetAt_TcVnRectangle_DINT : HRESULT
	VAR_INPUT
		ipContainer	:	ITcVnContainer;	(* Container with TcVnRectangle_DINT elements *)
		stElement	:	REFERENCE TO TcVnRectangle_DINT;	(* Returns the element at the specified index *)
		nIndex	:	ULINT;	(* Index of the requested element *)
		hrPrev	:	HRESULT;	(* HRESULT indicating the result of previous operations (If SUCCEEDED(hrPrev) equals false, no operation is executed.) *)
	END_VAR

END_FUNCTION

// Functions/Basic Container Operations/F_VN_GetAt/F_VN_GetAt_TcVnVector2_DINT

	{attribute 'TcIecLibraryType'}
	{attribute 'external_name' := 'F_VN_GetAt_TcVnVector2_DINT_GUID_E7C2B37B_70C4_3998_2382_4EB9E1DE7BCE'}
	(* Gets the TcVnVector2_DINT element at the specified index of the container. *)
	FUNCTION F_VN_GetAt_TcVnVector2_DINT : HRESULT
	VAR_INPUT
		ipContainer	:	ITcVnContainer;	(* Container with TcVnVector2_DINT elements *)
		aElement	:	REFERENCE TO TcVnVector2_DINT;	(* Returns the element at the specified index *)
		nIndex	:	ULINT;	(* Index of the requested element *)
		hrPrev	:	HRESULT;	(* HRESULT indicating the result of previous operations (If SUCCEEDED(hrPrev) equals false, no operation is executed.) *)
	END_VAR

END_FUNCTION

// Functions/Basic Container Operations/F_VN_GetAt/F_VN_GetAt_TcVnVector2_INT

	{attribute 'TcIecLibraryType'}
	{attribute 'external_name' := 'F_VN_GetAt_TcVnVector2_INT_GUID_70115FDC_19E9_3A1A_170B_469E5110F923'}
	(* Gets the TcVnVector2_INT element at the specified index of the container. *)
	FUNCTION F_VN_GetAt_TcVnVector2_INT : HRESULT
	VAR_INPUT
		ipContainer	:	ITcVnContainer;	(* Container with TcVnVector2_INT elements *)
		aElement	:	REFERENCE TO TcVnVector2_INT;	(* Returns the element at the specified index *)
		nIndex	:	ULINT;	(* Index of the requested element *)
		hrPrev	:	HRESULT;	(* HRESULT indicating the result of previous operations (If SUCCEEDED(hrPrev) equals false, no operation is executed.) *)
	END_VAR

END_FUNCTION

// Functions/Basic Container Operations/F_VN_GetAt/F_VN_GetAt_TcVnVector2_REAL

	{attribute 'TcIecLibraryType'}
	{attribute 'external_name' := 'F_VN_GetAt_TcVnVector2_REAL_GUID_934F0AF6_F9AB_31D8_2BAB_3B9DF8D54B4F'}
	(* Gets the TcVnVector2_REAL element at the specified index of the container. *)
	FUNCTION F_VN_GetAt_TcVnVector2_REAL : HRESULT
	VAR_INPUT
		ipContainer	:	ITcVnContainer;	(* Container with TcVnVector2_REAL elements *)
		aElement	:	REFERENCE TO TcVnVector2_REAL;	(* Returns the element at the specified index *)
		nIndex	:	ULINT;	(* Index of the requested element *)
		hrPrev	:	HRESULT;	(* HRESULT indicating the result of previous operations (If SUCCEEDED(hrPrev) equals false, no operation is executed.) *)
	END_VAR

END_FUNCTION

// Functions/Basic Container Operations/F_VN_GetAt/F_VN_GetAt_TcVnVector2_SINT

	{attribute 'TcIecLibraryType'}
	{attribute 'external_name' := 'F_VN_GetAt_TcVnVector2_SINT_GUID_A03F3DE8_F80B_3551_2585_744B19853183'}
	(* Gets the TcVnVector2_SINT element at the specified index of the container. *)
	FUNCTION F_VN_GetAt_TcVnVector2_SINT : HRESULT
	VAR_INPUT
		ipContainer	:	ITcVnContainer;	(* Container with TcVnVector2_SINT elements *)
		aElement	:	REFERENCE TO TcVnVector2_SINT;	(* Returns the element at the specified index *)
		nIndex	:	ULINT;	(* Index of the requested element *)
		hrPrev	:	HRESULT;	(* HRESULT indicating the result of previous operations (If SUCCEEDED(hrPrev) equals false, no operation is executed.) *)
	END_VAR

END_FUNCTION

// Functions/Basic Container Operations/F_VN_GetAt/F_VN_GetAt_TcVnVector2_UINT

	{attribute 'TcIecLibraryType'}
	{attribute 'external_name' := 'F_VN_GetAt_TcVnVector2_UINT_GUID_C1EC9D9A_FD3C_3A6B_078C_FD8ED4C33F35'}
	(* Gets the TcVnVector2_UINT element at the specified index of the container. *)
	FUNCTION F_VN_GetAt_TcVnVector2_UINT : HRESULT
	VAR_INPUT
		ipContainer	:	ITcVnContainer;	(* Container with TcVnVector2_UINT elements *)
		aElement	:	REFERENCE TO TcVnVector2_UINT;	(* Returns the element at the specified index *)
		nIndex	:	ULINT;	(* Index of the requested element *)
		hrPrev	:	HRESULT;	(* HRESULT indicating the result of previous operations (If SUCCEEDED(hrPrev) equals false, no operation is executed.) *)
	END_VAR

END_FUNCTION

// Functions/Basic Container Operations/F_VN_GetAt/F_VN_GetAt_TcVnVector2_USINT

	{attribute 'TcIecLibraryType'}
	{attribute 'external_name' := 'F_VN_GetAt_TcVnVector2_USINT_GUID_9151A628_DCD5_3225_06FF_C1BAF6F1DAB4'}
	(* Gets the TcVnVector2_USINT element at the specified index of the container. *)
	FUNCTION F_VN_GetAt_TcVnVector2_USINT : HRESULT
	VAR_INPUT
		ipContainer	:	ITcVnContainer;	(* Container with TcVnVector2_USINT elements *)
		aElement	:	REFERENCE TO TcVnVector2_USINT;	(* Returns the element at the specified index *)
		nIndex	:	ULINT;	(* Index of the requested element *)
		hrPrev	:	HRESULT;	(* HRESULT indicating the result of previous operations (If SUCCEEDED(hrPrev) equals false, no operation is executed.) *)
	END_VAR

END_FUNCTION

// Functions/Basic Container Operations/F_VN_GetAt/F_VN_GetAt_TcVnVector3_INT

	{attribute 'TcIecLibraryType'}
	{attribute 'external_name' := 'F_VN_GetAt_TcVnVector3_INT_GUID_5314E713_0BA0_360B_1F6E_965C93ECA65C'}
	(* Gets the TcVnVector3_INT element at the specified index of the container. *)
	FUNCTION F_VN_GetAt_TcVnVector3_INT : HRESULT
	VAR_INPUT
		ipContainer	:	ITcVnContainer;	(* Container with TcVnVector3_INT elements *)
		aElement	:	REFERENCE TO TcVnVector3_INT;	(* Returns the element at the specified index *)
		nIndex	:	ULINT;	(* Index of the requested element *)
		hrPrev	:	HRESULT;	(* HRESULT indicating the result of previous operations (If SUCCEEDED(hrPrev) equals false, no operation is executed.) *)
	END_VAR

END_FUNCTION

// Functions/Basic Container Operations/F_VN_GetAt/F_VN_GetAt_TcVnVector3_REAL

	{attribute 'TcIecLibraryType'}
	{attribute 'external_name' := 'F_VN_GetAt_TcVnVector3_REAL_GUID_EF583C7F_272D_3493_1464_1CEFBDA69B47'}
	(* Gets the TcVnVector3_REAL element at the specified index of the container. *)
	FUNCTION F_VN_GetAt_TcVnVector3_REAL : HRESULT
	VAR_INPUT
		ipContainer	:	ITcVnContainer;	(* Container with TcVnVector3_REAL elements *)
		aElement	:	REFERENCE TO TcVnVector3_REAL;	(* Returns the element at the specified index *)
		nIndex	:	ULINT;	(* Index of the requested element *)
		hrPrev	:	HRESULT;	(* HRESULT indicating the result of previous operations (If SUCCEEDED(hrPrev) equals false, no operation is executed.) *)
	END_VAR

END_FUNCTION

// Functions/Basic Container Operations/F_VN_GetAt/F_VN_GetAt_TcVnVector3_SINT

	{attribute 'TcIecLibraryType'}
	{attribute 'external_name' := 'F_VN_GetAt_TcVnVector3_SINT_GUID_F34424D2_DE97_3BDC_15BA_1766435215B5'}
	(* Gets the TcVnVector3_SINT element at the specified index of the container. *)
	FUNCTION F_VN_GetAt_TcVnVector3_SINT : HRESULT
	VAR_INPUT
		ipContainer	:	ITcVnContainer;	(* Container with TcVnVector3_SINT elements *)
		aElement	:	REFERENCE TO TcVnVector3_SINT;	(* Returns the element at the specified index *)
		nIndex	:	ULINT;	(* Index of the requested element *)
		hrPrev	:	HRESULT;	(* HRESULT indicating the result of previous operations (If SUCCEEDED(hrPrev) equals false, no operation is executed.) *)
	END_VAR

END_FUNCTION

// Functions/Basic Container Operations/F_VN_GetAt/F_VN_GetAt_TcVnVector3_UINT

	{attribute 'TcIecLibraryType'}
	{attribute 'external_name' := 'F_VN_GetAt_TcVnVector3_UINT_GUID_33DF0F8F_D380_3E26_387E_917D81CE9CB5'}
	(* Gets the TcVnVector3_UINT element at the specified index of the container. *)
	FUNCTION F_VN_GetAt_TcVnVector3_UINT : HRESULT
	VAR_INPUT
		ipContainer	:	ITcVnContainer;	(* Container with TcVnVector3_UINT elements *)
		aElement	:	REFERENCE TO TcVnVector3_UINT;	(* Returns the element at the specified index *)
		nIndex	:	ULINT;	(* Index of the requested element *)
		hrPrev	:	HRESULT;	(* HRESULT indicating the result of previous operations (If SUCCEEDED(hrPrev) equals false, no operation is executed.) *)
	END_VAR

END_FUNCTION

// Functions/Basic Container Operations/F_VN_GetAt/F_VN_GetAt_TcVnVector3_USINT

	{attribute 'TcIecLibraryType'}
	{attribute 'external_name' := 'F_VN_GetAt_TcVnVector3_USINT_GUID_6ABC03D4_28FD_3F19_2184_517A2F8C0024'}
	(* Gets the TcVnVector3_USINT element at the specified index of the container. *)
	FUNCTION F_VN_GetAt_TcVnVector3_USINT : HRESULT
	VAR_INPUT
		ipContainer	:	ITcVnContainer;	(* Container with TcVnVector3_USINT elements *)
		aElement	:	REFERENCE TO TcVnVector3_USINT;	(* Returns the element at the specified index *)
		nIndex	:	ULINT;	(* Index of the requested element *)
		hrPrev	:	HRESULT;	(* HRESULT indicating the result of previous operations (If SUCCEEDED(hrPrev) equals false, no operation is executed.) *)
	END_VAR

END_FUNCTION

// Functions/Basic Container Operations/F_VN_GetAt/F_VN_GetAt_TcVnVector4_DINT

	{attribute 'TcIecLibraryType'}
	{attribute 'external_name' := 'F_VN_GetAt_TcVnVector4_DINT_GUID_EA0F74F7_D6EB_3664_248F_3C7B9C7DD045'}
	(* Gets the TcVnVector4_DINT element at the specified index of the container. *)
	FUNCTION F_VN_GetAt_TcVnVector4_DINT : HRESULT
	VAR_INPUT
		ipContainer	:	ITcVnContainer;	(* Container with TcVnVector4_DINT elements *)
		aElement	:	REFERENCE TO TcVnVector4_DINT;	(* Returns the element at the specified index *)
		nIndex	:	ULINT;	(* Index of the requested element *)
		hrPrev	:	HRESULT;	(* HRESULT indicating the result of previous operations (If SUCCEEDED(hrPrev) equals false, no operation is executed.) *)
	END_VAR

END_FUNCTION

// Functions/Basic Container Operations/F_VN_GetAt/F_VN_GetAt_TcVnVector4_INT

	{attribute 'TcIecLibraryType'}
	{attribute 'external_name' := 'F_VN_GetAt_TcVnVector4_INT_GUID_6B938A06_FC67_3C66_1CCB_99CA533A0F62'}
	(* Gets the TcVnVector4_INT element at the specified index of the container. *)
	FUNCTION F_VN_GetAt_TcVnVector4_INT : HRESULT
	VAR_INPUT
		ipContainer	:	ITcVnContainer;	(* Container with TcVnVector4_INT elements *)
		aElement	:	REFERENCE TO TcVnVector4_INT;	(* Returns the element at the specified index *)
		nIndex	:	ULINT;	(* Index of the requested element *)
		hrPrev	:	HRESULT;	(* HRESULT indicating the result of previous operations (If SUCCEEDED(hrPrev) equals false, no operation is executed.) *)
	END_VAR

END_FUNCTION

// Functions/Basic Container Operations/F_VN_GetAt/F_VN_GetAt_TcVnVector4_LREAL

	{attribute 'TcIecLibraryType'}
	{attribute 'external_name' := 'F_VN_GetAt_TcVnVector4_LREAL_GUID_C3C98E2A_44FB_36C5_24B6_BADEB04CBA29'}
	(* Gets the TcVnVector4_LREAL element at the specified index of the container. *)
	FUNCTION F_VN_GetAt_TcVnVector4_LREAL : HRESULT
	VAR_INPUT
		ipContainer	:	ITcVnContainer;	(* Container with TcVnVector4_LREAL elements *)
		aElement	:	REFERENCE TO TcVnVector4_LREAL;	(* Returns the element at the specified index *)
		nIndex	:	ULINT;	(* Index of the requested element *)
		hrPrev	:	HRESULT;	(* HRESULT indicating the result of previous operations (If SUCCEEDED(hrPrev) equals false, no operation is executed.) *)
	END_VAR

END_FUNCTION

// Functions/Basic Container Operations/F_VN_GetAt/F_VN_GetAt_TcVnVector4_SINT

	{attribute 'TcIecLibraryType'}
	{attribute 'external_name' := 'F_VN_GetAt_TcVnVector4_SINT_GUID_BB245398_13B3_3BF4_1357_8161B2BD5E05'}
	(* Gets the TcVnVector4_SINT element at the specified index of the container. *)
	FUNCTION F_VN_GetAt_TcVnVector4_SINT : HRESULT
	VAR_INPUT
		ipContainer	:	ITcVnContainer;	(* Container with TcVnVector4_SINT elements *)
		aElement	:	REFERENCE TO TcVnVector4_SINT;	(* Returns the element at the specified index *)
		nIndex	:	ULINT;	(* Index of the requested element *)
		hrPrev	:	HRESULT;	(* HRESULT indicating the result of previous operations (If SUCCEEDED(hrPrev) equals false, no operation is executed.) *)
	END_VAR

END_FUNCTION

// Functions/Basic Container Operations/F_VN_GetAt/F_VN_GetAt_TcVnVector4_UINT

	{attribute 'TcIecLibraryType'}
	{attribute 'external_name' := 'F_VN_GetAt_TcVnVector4_UINT_GUID_3D08AD04_885D_3AE5_26C0_0AA5E2D37788'}
	(* Gets the TcVnVector4_UINT element at the specified index of the container. *)
	FUNCTION F_VN_GetAt_TcVnVector4_UINT : HRESULT
	VAR_INPUT
		ipContainer	:	ITcVnContainer;	(* Container with TcVnVector4_UINT elements *)
		aElement	:	REFERENCE TO TcVnVector4_UINT;	(* Returns the element at the specified index *)
		nIndex	:	ULINT;	(* Index of the requested element *)
		hrPrev	:	HRESULT;	(* HRESULT indicating the result of previous operations (If SUCCEEDED(hrPrev) equals false, no operation is executed.) *)
	END_VAR

END_FUNCTION

// Functions/Basic Container Operations/F_VN_GetAt/F_VN_GetAt_TcVnVector4_USINT

	{attribute 'TcIecLibraryType'}
	{attribute 'external_name' := 'F_VN_GetAt_TcVnVector4_USINT_GUID_578E5B9E_2C40_3A76_3D53_BD5F2823DEA9'}
	(* Gets the TcVnVector4_USINT element at the specified index of the container. *)
	FUNCTION F_VN_GetAt_TcVnVector4_USINT : HRESULT
	VAR_INPUT
		ipContainer	:	ITcVnContainer;	(* Container with TcVnVector4_USINT elements *)
		aElement	:	REFERENCE TO TcVnVector4_USINT;	(* Returns the element at the specified index *)
		nIndex	:	ULINT;	(* Index of the requested element *)
		hrPrev	:	HRESULT;	(* HRESULT indicating the result of previous operations (If SUCCEEDED(hrPrev) equals false, no operation is executed.) *)
	END_VAR

END_FUNCTION

// Functions/Basic Container Operations/F_VN_GetAt/F_VN_GetAt_UDINT

	{attribute 'TcIecLibraryType'}
	{attribute 'external_name' := 'F_VN_GetAt_UDINT_GUID_58551719_6068_3651_1231_574E227F0984'}
	(* Gets the UDINT element at the specified index of the container. *)
	FUNCTION F_VN_GetAt_UDINT : HRESULT
	VAR_INPUT
		ipContainer	:	ITcVnContainer;	(* Container with UDINT elements *)
		nElement	:	REFERENCE TO UDINT;	(* Returns the element at the specified index *)
		nIndex	:	ULINT;	(* Index of the requested element *)
		hrPrev	:	HRESULT;	(* HRESULT indicating the result of previous operations (If SUCCEEDED(hrPrev) equals false, no operation is executed.) *)
	END_VAR

END_FUNCTION

// Functions/Basic Container Operations/F_VN_GetAt/F_VN_GetAt_UINT

	{attribute 'TcIecLibraryType'}
	{attribute 'external_name' := 'F_VN_GetAt_UINT_GUID_33355A0E_717D_3A70_343D_FDEF92E0E58C'}
	(* Gets the UINT element at the specified index of the container. *)
	FUNCTION F_VN_GetAt_UINT : HRESULT
	VAR_INPUT
		ipContainer	:	ITcVnContainer;	(* Container with UINT elements *)
		nElement	:	REFERENCE TO UINT;	(* Returns the element at the specified index *)
		nIndex	:	ULINT;	(* Index of the requested element *)
		hrPrev	:	HRESULT;	(* HRESULT indicating the result of previous operations (If SUCCEEDED(hrPrev) equals false, no operation is executed.) *)
	END_VAR

END_FUNCTION

// Functions/Basic Container Operations/F_VN_GetAt/F_VN_GetAt_ULINT

	{attribute 'TcIecLibraryType'}
	{attribute 'external_name' := 'F_VN_GetAt_ULINT_GUID_5B72C1CA_E9B3_3B06_13F4_872ECAA28495'}
	(* Gets the ULINT element at the specified index of the container. *)
	FUNCTION F_VN_GetAt_ULINT : HRESULT
	VAR_INPUT
		ipContainer	:	ITcVnContainer;	(* Container with ULINT elements *)
		nElement	:	REFERENCE TO ULINT;	(* Returns the element at the specified index *)
		nIndex	:	ULINT;	(* Index of the requested element *)
		hrPrev	:	HRESULT;	(* HRESULT indicating the result of previous operations (If SUCCEEDED(hrPrev) equals false, no operation is executed.) *)
	END_VAR

END_FUNCTION

// Functions/Basic Container Operations/F_VN_GetAt/F_VN_GetAt_USINT

	{attribute 'TcIecLibraryType'}
	{attribute 'external_name' := 'F_VN_GetAt_USINT_GUID_D98B5672_7560_38E1_03A6_75AC2CA9D484'}
	(* Gets the USINT element at the specified index of the container. *)
	FUNCTION F_VN_GetAt_USINT : HRESULT
	VAR_INPUT
		ipContainer	:	ITcVnContainer;	(* Container with USINT elements *)
		nElement	:	REFERENCE TO USINT;	(* Returns the element at the specified index *)
		nIndex	:	ULINT;	(* Index of the requested element *)
		hrPrev	:	HRESULT;	(* HRESULT indicating the result of previous operations (If SUCCEEDED(hrPrev) equals false, no operation is executed.) *)
	END_VAR

END_FUNCTION

// Functions/Basic Container Operations/F_VN_InsertIntoContainer/F_VN_InsertIntoContainer_ITcVnContainer

	{attribute 'TcIecLibraryType'}
	{attribute 'external_name' := 'F_VN_InsertIntoContainer_ITcVnContainer_GUID_41C95B3F_A3FB_3603_21B3_C7F2865D3F76'}
	(* Insert an element (or a range of elements) into a container before the specified position. *)
	FUNCTION F_VN_InsertIntoContainer_ITcVnContainer : HRESULT
	VAR_INPUT
		ipElement	:	ITcVnContainer;	(* Single element to insert into ipContainer or container with several elements *)
		ipContainer	:	ITcVnContainer;	(* Container in which to insert the element *)
		nIndex	:	ULINT;	(* Position, before which the element will be inserted *)
		hrPrev	:	HRESULT;	(* HRESULT indicating the result of previous operations (If SUCCEEDED(hrPrev) equals false, no operation is executed.) *)
	END_VAR

END_FUNCTION

// Functions/Basic Container Operations/F_VN_InsertIntoContainer/F_VN_InsertIntoContainer_ITcVnForwardIterator

	{attribute 'TcIecLibraryType'}
	{attribute 'external_name' := 'F_VN_InsertIntoContainer_ITcVnForwardIterator_GUID_1CB7BC98_F0EE_30A1_259C_32EBCD627F75'}
	(* Insert an element (represented by an iterator) into a container before the specified position. *)
	FUNCTION F_VN_InsertIntoContainer_ITcVnForwardIterator : HRESULT
	VAR_INPUT
		ipElement	:	ITcVnForwardIterator;	(* Single element to insert into ipContainer *)
		ipContainer	:	ITcVnContainer;	(* Container in which to insert the element *)
		nIndex	:	ULINT;	(* Position, before which the element will be inserted *)
		hrPrev	:	HRESULT;	(* HRESULT indicating the result of previous operations (If SUCCEEDED(hrPrev) equals false, no operation is executed.) *)
	END_VAR

END_FUNCTION

// Functions/Basic Container Operations/F_VN_InsertIntoContainer/F_VN_InsertIntoContainer_DINT

	{attribute 'TcIecLibraryType'}
	{attribute 'external_name' := 'F_VN_InsertIntoContainer_DINT_GUID_73B53AF7_64C7_3533_33BF_2473D8A45673'}
	(* Insert an element of type DINT into a container before the specified position. *)
	FUNCTION F_VN_InsertIntoContainer_DINT : HRESULT
	VAR_INPUT
		nElement	:	DINT;	(* Single element to insert into ipContainer *)
		ipContainer	:	ITcVnContainer;	(* Container in which to insert the element *)
		nIndex	:	ULINT;	(* Position, before which the element will be inserted *)
		hrPrev	:	HRESULT;	(* HRESULT indicating the result of previous operations (If SUCCEEDED(hrPrev) equals false, no operation is executed.) *)
	END_VAR

END_FUNCTION

// Functions/Basic Container Operations/F_VN_InsertIntoContainer/F_VN_InsertIntoContainer_INT

	{attribute 'TcIecLibraryType'}
	{attribute 'external_name' := 'F_VN_InsertIntoContainer_INT_GUID_8B917B5E_2BF7_3174_2464_5D13E2572D53'}
	(* Insert an element of type INT into a container before the specified position. *)
	FUNCTION F_VN_InsertIntoContainer_INT : HRESULT
	VAR_INPUT
		nElement	:	INT;	(* Single element to insert into ipContainer *)
		ipContainer	:	ITcVnContainer;	(* Container in which to insert the element *)
		nIndex	:	ULINT;	(* Position, before which the element will be inserted *)
		hrPrev	:	HRESULT;	(* HRESULT indicating the result of previous operations (If SUCCEEDED(hrPrev) equals false, no operation is executed.) *)
	END_VAR

END_FUNCTION

// Functions/Basic Container Operations/F_VN_InsertIntoContainer/F_VN_InsertIntoContainer_LREAL

	{attribute 'TcIecLibraryType'}
	{attribute 'external_name' := 'F_VN_InsertIntoContainer_LREAL_GUID_EEADD051_7813_3477_299F_4762ACAD308D'}
	(* Insert an element of type LREAL into a container before the specified position. *)
	FUNCTION F_VN_InsertIntoContainer_LREAL : HRESULT
	VAR_INPUT
		fElement	:	LREAL;	(* Single element to insert into ipContainer *)
		ipContainer	:	ITcVnContainer;	(* Container in which to insert the element *)
		nIndex	:	ULINT;	(* Position, before which the element will be inserted *)
		hrPrev	:	HRESULT;	(* HRESULT indicating the result of previous operations (If SUCCEEDED(hrPrev) equals false, no operation is executed.) *)
	END_VAR

END_FUNCTION

// Functions/Basic Container Operations/F_VN_InsertIntoContainer/F_VN_InsertIntoContainer_REAL

	{attribute 'TcIecLibraryType'}
	{attribute 'external_name' := 'F_VN_InsertIntoContainer_REAL_GUID_A2B306BC_8AA3_35A8_3D84_291126C7545B'}
	(* Insert an element of type REAL into a container before the specified position. *)
	FUNCTION F_VN_InsertIntoContainer_REAL : HRESULT
	VAR_INPUT
		fElement	:	REAL;	(* Single element to insert into ipContainer *)
		ipContainer	:	ITcVnContainer;	(* Container in which to insert the element *)
		nIndex	:	ULINT;	(* Position, before which the element will be inserted *)
		hrPrev	:	HRESULT;	(* HRESULT indicating the result of previous operations (If SUCCEEDED(hrPrev) equals false, no operation is executed.) *)
	END_VAR

END_FUNCTION

// Functions/Basic Container Operations/F_VN_InsertIntoContainer/F_VN_InsertIntoContainer_SINT

	{attribute 'TcIecLibraryType'}
	{attribute 'external_name' := 'F_VN_InsertIntoContainer_SINT_GUID_403DD2CE_19C6_32C3_3367_EF0932EE5D29'}
	(* Insert an element of type SINT into a container before the specified position. *)
	FUNCTION F_VN_InsertIntoContainer_SINT : HRESULT
	VAR_INPUT
		nElement	:	SINT;	(* Single element to insert into ipContainer *)
		ipContainer	:	ITcVnContainer;	(* Container in which to insert the element *)
		nIndex	:	ULINT;	(* Position, before which the element will be inserted *)
		hrPrev	:	HRESULT;	(* HRESULT indicating the result of previous operations (If SUCCEEDED(hrPrev) equals false, no operation is executed.) *)
	END_VAR

END_FUNCTION

// Functions/Basic Container Operations/F_VN_InsertIntoContainer/F_VN_InsertIntoContainer_TcVnDMatch

	{attribute 'TcIecLibraryType'}
	{attribute 'external_name' := 'F_VN_InsertIntoContainer_TcVnDMatch_GUID_FE9D2741_0BB4_3D98_15F9_6F5BE6F89A13'}
	(* Insert an element of type TcVnDMatch into a container before the specified position. *)
	FUNCTION F_VN_InsertIntoContainer_TcVnDMatch : HRESULT
	VAR_INPUT
		stElement	:	REFERENCE TO TcVnDMatch;	(* Single element to insert into ipContainer *)
		ipContainer	:	ITcVnContainer;	(* Container in which to insert the element *)
		nIndex	:	ULINT;	(* Position, before which the element will be inserted *)
		hrPrev	:	HRESULT;	(* HRESULT indicating the result of previous operations (If SUCCEEDED(hrPrev) equals false, no operation is executed.) *)
	END_VAR

END_FUNCTION

// Functions/Basic Container Operations/F_VN_InsertIntoContainer/F_VN_InsertIntoContainer_TcVnKeyPoint

	{attribute 'TcIecLibraryType'}
	{attribute 'external_name' := 'F_VN_InsertIntoContainer_TcVnKeyPoint_GUID_2A31F0C2_C9DF_303C_1813_998AF65B057D'}
	(* Insert an element of type TcVnKeyPoint into a container before the specified position. *)
	FUNCTION F_VN_InsertIntoContainer_TcVnKeyPoint : HRESULT
	VAR_INPUT
		stElement	:	REFERENCE TO TcVnKeyPoint;	(* Single element to insert into ipContainer *)
		ipContainer	:	ITcVnContainer;	(* Container in which to insert the element *)
		nIndex	:	ULINT;	(* Position, before which the element will be inserted *)
		hrPrev	:	HRESULT;	(* HRESULT indicating the result of previous operations (If SUCCEEDED(hrPrev) equals false, no operation is executed.) *)
	END_VAR

END_FUNCTION

// Functions/Basic Container Operations/F_VN_InsertIntoContainer/F_VN_InsertIntoContainer_TcVnPoint2_DINT

	{attribute 'TcIecLibraryType'}
	{attribute 'external_name' := 'F_VN_InsertIntoContainer_TcVnPoint2_DINT_GUID_695C020D_F65C_36AD_0C20_4D36BDE70083'}
	(* Insert an element of type TcVnPoint2_DINT into a container before the specified position. *)
	FUNCTION F_VN_InsertIntoContainer_TcVnPoint2_DINT : HRESULT
	VAR_INPUT
		aElement	:	REFERENCE TO TcVnPoint2_DINT;	(* Single element to insert into ipContainer *)
		ipContainer	:	ITcVnContainer;	(* Container in which to insert the element *)
		nIndex	:	ULINT;	(* Position, before which the element will be inserted *)
		hrPrev	:	HRESULT;	(* HRESULT indicating the result of previous operations (If SUCCEEDED(hrPrev) equals false, no operation is executed.) *)
	END_VAR

END_FUNCTION

// Functions/Basic Container Operations/F_VN_InsertIntoContainer/F_VN_InsertIntoContainer_TcVnPoint2_LREAL

	{attribute 'TcIecLibraryType'}
	{attribute 'external_name' := 'F_VN_InsertIntoContainer_TcVnPoint2_LREAL_GUID_932769FA_DE0B_3C85_1AF1_7BBE0783DC31'}
	(* Insert an element of type TcVnPoint2_LREAL into a container before the specified position. *)
	FUNCTION F_VN_InsertIntoContainer_TcVnPoint2_LREAL : HRESULT
	VAR_INPUT
		aElement	:	REFERENCE TO TcVnPoint2_LREAL;	(* Single element to insert into ipContainer *)
		ipContainer	:	ITcVnContainer;	(* Container in which to insert the element *)
		nIndex	:	ULINT;	(* Position, before which the element will be inserted *)
		hrPrev	:	HRESULT;	(* HRESULT indicating the result of previous operations (If SUCCEEDED(hrPrev) equals false, no operation is executed.) *)
	END_VAR

END_FUNCTION

// Functions/Basic Container Operations/F_VN_InsertIntoContainer/F_VN_InsertIntoContainer_TcVnPoint2_REAL

	{attribute 'TcIecLibraryType'}
	{attribute 'external_name' := 'F_VN_InsertIntoContainer_TcVnPoint2_REAL_GUID_EE6A7FEC_81D0_3406_3115_C930F8F9A783'}
	(* Insert an element of type TcVnPoint2_REAL into a container before the specified position. *)
	FUNCTION F_VN_InsertIntoContainer_TcVnPoint2_REAL : HRESULT
	VAR_INPUT
		aElement	:	REFERENCE TO TcVnPoint2_REAL;	(* Single element to insert into ipContainer *)
		ipContainer	:	ITcVnContainer;	(* Container in which to insert the element *)
		nIndex	:	ULINT;	(* Position, before which the element will be inserted *)
		hrPrev	:	HRESULT;	(* HRESULT indicating the result of previous operations (If SUCCEEDED(hrPrev) equals false, no operation is executed.) *)
	END_VAR

END_FUNCTION

// Functions/Basic Container Operations/F_VN_InsertIntoContainer/F_VN_InsertIntoContainer_TcVnPoint3_LREAL

	{attribute 'TcIecLibraryType'}
	{attribute 'external_name' := 'F_VN_InsertIntoContainer_TcVnPoint3_LREAL_GUID_9B66BA24_FA57_3C14_3C5A_03925DE703D3'}
	(* Insert an element of type TcVnPoint3_LREAL into a container before the specified position. *)
	FUNCTION F_VN_InsertIntoContainer_TcVnPoint3_LREAL : HRESULT
	VAR_INPUT
		aElement	:	REFERENCE TO TcVnPoint3_LREAL;	(* Single element to insert into ipContainer *)
		ipContainer	:	ITcVnContainer;	(* Container in which to insert the element *)
		nIndex	:	ULINT;	(* Position, before which the element will be inserted *)
		hrPrev	:	HRESULT;	(* HRESULT indicating the result of previous operations (If SUCCEEDED(hrPrev) equals false, no operation is executed.) *)
	END_VAR

END_FUNCTION

// Functions/Basic Container Operations/F_VN_InsertIntoContainer/F_VN_InsertIntoContainer_TcVnPoint3_REAL

	{attribute 'TcIecLibraryType'}
	{attribute 'external_name' := 'F_VN_InsertIntoContainer_TcVnPoint3_REAL_GUID_FA76F7B1_C375_329F_185C_CEE667FBC135'}
	(* Insert an element of type TcVnPoint3_REAL into a container before the specified position. *)
	FUNCTION F_VN_InsertIntoContainer_TcVnPoint3_REAL : HRESULT
	VAR_INPUT
		aElement	:	REFERENCE TO TcVnPoint3_REAL;	(* Single element to insert into ipContainer *)
		ipContainer	:	ITcVnContainer;	(* Container in which to insert the element *)
		nIndex	:	ULINT;	(* Position, before which the element will be inserted *)
		hrPrev	:	HRESULT;	(* HRESULT indicating the result of previous operations (If SUCCEEDED(hrPrev) equals false, no operation is executed.) *)
	END_VAR

END_FUNCTION

// Functions/Basic Container Operations/F_VN_InsertIntoContainer/F_VN_InsertIntoContainer_TcVnRectangle_DINT

	{attribute 'TcIecLibraryType'}
	{attribute 'external_name' := 'F_VN_InsertIntoContainer_TcVnRectangle_DINT_GUID_F129AF62_3045_3CC1_20F3_8A613580F7AD'}
	(* Insert an element of type TcVnRectangle_DINT into a container before the specified position. *)
	FUNCTION F_VN_InsertIntoContainer_TcVnRectangle_DINT : HRESULT
	VAR_INPUT
		stElement	:	REFERENCE TO TcVnRectangle_DINT;	(* Single element to insert into ipContainer *)
		ipContainer	:	ITcVnContainer;	(* Container in which to insert the element *)
		nIndex	:	ULINT;	(* Position, before which the element will be inserted *)
		hrPrev	:	HRESULT;	(* HRESULT indicating the result of previous operations (If SUCCEEDED(hrPrev) equals false, no operation is executed.) *)
	END_VAR

END_FUNCTION

// Functions/Basic Container Operations/F_VN_InsertIntoContainer/F_VN_InsertIntoContainer_TcVnVector2_DINT

	{attribute 'TcIecLibraryType'}
	{attribute 'external_name' := 'F_VN_InsertIntoContainer_TcVnVector2_DINT_GUID_0AC6F463_7496_3D8F_25B0_46CD51B9B8E3'}
	(* Insert an element of type TcVnVector2_DINT into a container before the specified position. *)
	FUNCTION F_VN_InsertIntoContainer_TcVnVector2_DINT : HRESULT
	VAR_INPUT
		aElement	:	REFERENCE TO TcVnVector2_DINT;	(* Single element to insert into ipContainer *)
		ipContainer	:	ITcVnContainer;	(* Container in which to insert the element *)
		nIndex	:	ULINT;	(* Position, before which the element will be inserted *)
		hrPrev	:	HRESULT;	(* HRESULT indicating the result of previous operations (If SUCCEEDED(hrPrev) equals false, no operation is executed.) *)
	END_VAR

END_FUNCTION

// Functions/Basic Container Operations/F_VN_InsertIntoContainer/F_VN_InsertIntoContainer_TcVnVector2_INT

	{attribute 'TcIecLibraryType'}
	{attribute 'external_name' := 'F_VN_InsertIntoContainer_TcVnVector2_INT_GUID_75E4ECBD_A466_3301_1A51_F9BE5833FD89'}
	(* Insert an element of type TcVnVector2_INT into a container before the specified position. *)
	FUNCTION F_VN_InsertIntoContainer_TcVnVector2_INT : HRESULT
	VAR_INPUT
		aElement	:	REFERENCE TO TcVnVector2_INT;	(* Single element to insert into ipContainer *)
		ipContainer	:	ITcVnContainer;	(* Container in which to insert the element *)
		nIndex	:	ULINT;	(* Position, before which the element will be inserted *)
		hrPrev	:	HRESULT;	(* HRESULT indicating the result of previous operations (If SUCCEEDED(hrPrev) equals false, no operation is executed.) *)
	END_VAR

END_FUNCTION

// Functions/Basic Container Operations/F_VN_InsertIntoContainer/F_VN_InsertIntoContainer_TcVnVector2_REAL

	{attribute 'TcIecLibraryType'}
	{attribute 'external_name' := 'F_VN_InsertIntoContainer_TcVnVector2_REAL_GUID_7B54DC15_EABD_3A05_32E0_9850B5AB7B96'}
	(* Insert an element of type TcVnVector2_REAL into a container before the specified position. *)
	FUNCTION F_VN_InsertIntoContainer_TcVnVector2_REAL : HRESULT
	VAR_INPUT
		aElement	:	REFERENCE TO TcVnVector2_REAL;	(* Single element to insert into ipContainer *)
		ipContainer	:	ITcVnContainer;	(* Container in which to insert the element *)
		nIndex	:	ULINT;	(* Position, before which the element will be inserted *)
		hrPrev	:	HRESULT;	(* HRESULT indicating the result of previous operations (If SUCCEEDED(hrPrev) equals false, no operation is executed.) *)
	END_VAR

END_FUNCTION

// Functions/Basic Container Operations/F_VN_InsertIntoContainer/F_VN_InsertIntoContainer_TcVnVector2_SINT

	{attribute 'TcIecLibraryType'}
	{attribute 'external_name' := 'F_VN_InsertIntoContainer_TcVnVector2_SINT_GUID_2006850F_526D_35F1_0444_F334E2A5336F'}
	(* Insert an element of type TcVnVector2_SINT into a container before the specified position. *)
	FUNCTION F_VN_InsertIntoContainer_TcVnVector2_SINT : HRESULT
	VAR_INPUT
		aElement	:	REFERENCE TO TcVnVector2_SINT;	(* Single element to insert into ipContainer *)
		ipContainer	:	ITcVnContainer;	(* Container in which to insert the element *)
		nIndex	:	ULINT;	(* Position, before which the element will be inserted *)
		hrPrev	:	HRESULT;	(* HRESULT indicating the result of previous operations (If SUCCEEDED(hrPrev) equals false, no operation is executed.) *)
	END_VAR

END_FUNCTION

// Functions/Basic Container Operations/F_VN_InsertIntoContainer/F_VN_InsertIntoContainer_TcVnVector2_UINT

	{attribute 'TcIecLibraryType'}
	{attribute 'external_name' := 'F_VN_InsertIntoContainer_TcVnVector2_UINT_GUID_84DF90CF_BC15_3EA1_2E64_1A0488B06748'}
	(* Insert an element of type TcVnVector2_UINT into a container before the specified position. *)
	FUNCTION F_VN_InsertIntoContainer_TcVnVector2_UINT : HRESULT
	VAR_INPUT
		aElement	:	REFERENCE TO TcVnVector2_UINT;	(* Single element to insert into ipContainer *)
		ipContainer	:	ITcVnContainer;	(* Container in which to insert the element *)
		nIndex	:	ULINT;	(* Position, before which the element will be inserted *)
		hrPrev	:	HRESULT;	(* HRESULT indicating the result of previous operations (If SUCCEEDED(hrPrev) equals false, no operation is executed.) *)
	END_VAR

END_FUNCTION

// Functions/Basic Container Operations/F_VN_InsertIntoContainer/F_VN_InsertIntoContainer_TcVnVector2_USINT

	{attribute 'TcIecLibraryType'}
	{attribute 'external_name' := 'F_VN_InsertIntoContainer_TcVnVector2_USINT_GUID_070D1FA2_5478_3111_11F0_75D82B0478D6'}
	(* Insert an element of type TcVnVector2_USINT into a container before the specified position. *)
	FUNCTION F_VN_InsertIntoContainer_TcVnVector2_USINT : HRESULT
	VAR_INPUT
		aElement	:	REFERENCE TO TcVnVector2_USINT;	(* Single element to insert into ipContainer *)
		ipContainer	:	ITcVnContainer;	(* Container in which to insert the element *)
		nIndex	:	ULINT;	(* Position, before which the element will be inserted *)
		hrPrev	:	HRESULT;	(* HRESULT indicating the result of previous operations (If SUCCEEDED(hrPrev) equals false, no operation is executed.) *)
	END_VAR

END_FUNCTION

// Functions/Basic Container Operations/F_VN_InsertIntoContainer/F_VN_InsertIntoContainer_TcVnVector3_INT

	{attribute 'TcIecLibraryType'}
	{attribute 'external_name' := 'F_VN_InsertIntoContainer_TcVnVector3_INT_GUID_C9F40601_6E2F_31A1_200E_D2AED4B3AB34'}
	(* Insert an element of type TcVnVector3_INT into a container before the specified position. *)
	FUNCTION F_VN_InsertIntoContainer_TcVnVector3_INT : HRESULT
	VAR_INPUT
		aElement	:	REFERENCE TO TcVnVector3_INT;	(* Single element to insert into ipContainer *)
		ipContainer	:	ITcVnContainer;	(* Container in which to insert the element *)
		nIndex	:	ULINT;	(* Position, before which the element will be inserted *)
		hrPrev	:	HRESULT;	(* HRESULT indicating the result of previous operations (If SUCCEEDED(hrPrev) equals false, no operation is executed.) *)
	END_VAR

END_FUNCTION

// Functions/Basic Container Operations/F_VN_InsertIntoContainer/F_VN_InsertIntoContainer_TcVnVector3_REAL

	{attribute 'TcIecLibraryType'}
	{attribute 'external_name' := 'F_VN_InsertIntoContainer_TcVnVector3_REAL_GUID_E204F378_4844_39B5_2995_6A1A79AA8576'}
	(* Insert an element of type TcVnVector3_REAL into a container before the specified position. *)
	FUNCTION F_VN_InsertIntoContainer_TcVnVector3_REAL : HRESULT
	VAR_INPUT
		aElement	:	REFERENCE TO TcVnVector3_REAL;	(* Single element to insert into ipContainer *)
		ipContainer	:	ITcVnContainer;	(* Container in which to insert the element *)
		nIndex	:	ULINT;	(* Position, before which the element will be inserted *)
		hrPrev	:	HRESULT;	(* HRESULT indicating the result of previous operations (If SUCCEEDED(hrPrev) equals false, no operation is executed.) *)
	END_VAR

END_FUNCTION

// Functions/Basic Container Operations/F_VN_InsertIntoContainer/F_VN_InsertIntoContainer_TcVnVector3_SINT

	{attribute 'TcIecLibraryType'}
	{attribute 'external_name' := 'F_VN_InsertIntoContainer_TcVnVector3_SINT_GUID_F0A80B6D_32B7_38B6_1CF0_23E272AB8EB9'}
	(* Insert an element of type TcVnVector3_SINT into a container before the specified position. *)
	FUNCTION F_VN_InsertIntoContainer_TcVnVector3_SINT : HRESULT
	VAR_INPUT
		aElement	:	REFERENCE TO TcVnVector3_SINT;	(* Single element to insert into ipContainer *)
		ipContainer	:	ITcVnContainer;	(* Container in which to insert the element *)
		nIndex	:	ULINT;	(* Position, before which the element will be inserted *)
		hrPrev	:	HRESULT;	(* HRESULT indicating the result of previous operations (If SUCCEEDED(hrPrev) equals false, no operation is executed.) *)
	END_VAR

END_FUNCTION

// Functions/Basic Container Operations/F_VN_InsertIntoContainer/F_VN_InsertIntoContainer_TcVnVector3_UINT

	{attribute 'TcIecLibraryType'}
	{attribute 'external_name' := 'F_VN_InsertIntoContainer_TcVnVector3_UINT_GUID_C7E06659_8BFB_3F8B_2A36_820F8A3A1636'}
	(* Insert an element of type TcVnVector3_UINT into a container before the specified position. *)
	FUNCTION F_VN_InsertIntoContainer_TcVnVector3_UINT : HRESULT
	VAR_INPUT
		aElement	:	REFERENCE TO TcVnVector3_UINT;	(* Single element to insert into ipContainer *)
		ipContainer	:	ITcVnContainer;	(* Container in which to insert the element *)
		nIndex	:	ULINT;	(* Position, before which the element will be inserted *)
		hrPrev	:	HRESULT;	(* HRESULT indicating the result of previous operations (If SUCCEEDED(hrPrev) equals false, no operation is executed.) *)
	END_VAR

END_FUNCTION

// Functions/Basic Container Operations/F_VN_InsertIntoContainer/F_VN_InsertIntoContainer_TcVnVector3_USINT

	{attribute 'TcIecLibraryType'}
	{attribute 'external_name' := 'F_VN_InsertIntoContainer_TcVnVector3_USINT_GUID_AEB41AEB_E7C8_35ED_08D9_EE43B4444BC8'}
	(* Insert an element of type TcVnVector3_USINT into a container before the specified position. *)
	FUNCTION F_VN_InsertIntoContainer_TcVnVector3_USINT : HRESULT
	VAR_INPUT
		aElement	:	REFERENCE TO TcVnVector3_USINT;	(* Single element to insert into ipContainer *)
		ipContainer	:	ITcVnContainer;	(* Container in which to insert the element *)
		nIndex	:	ULINT;	(* Position, before which the element will be inserted *)
		hrPrev	:	HRESULT;	(* HRESULT indicating the result of previous operations (If SUCCEEDED(hrPrev) equals false, no operation is executed.) *)
	END_VAR

END_FUNCTION

// Functions/Basic Container Operations/F_VN_InsertIntoContainer/F_VN_InsertIntoContainer_TcVnVector4_DINT

	{attribute 'TcIecLibraryType'}
	{attribute 'external_name' := 'F_VN_InsertIntoContainer_TcVnVector4_DINT_GUID_D62F1BDB_734C_3DE3_196A_06FD075FDB6E'}
	(* Insert an element of type TcVnVector4_DINT into a container before the specified position. *)
	FUNCTION F_VN_InsertIntoContainer_TcVnVector4_DINT : HRESULT
	VAR_INPUT
		aElement	:	REFERENCE TO TcVnVector4_DINT;	(* Single element to insert into ipContainer *)
		ipContainer	:	ITcVnContainer;	(* Container in which to insert the element *)
		nIndex	:	ULINT;	(* Position, before which the element will be inserted *)
		hrPrev	:	HRESULT;	(* HRESULT indicating the result of previous operations (If SUCCEEDED(hrPrev) equals false, no operation is executed.) *)
	END_VAR

END_FUNCTION

// Functions/Basic Container Operations/F_VN_InsertIntoContainer/F_VN_InsertIntoContainer_TcVnVector4_INT

	{attribute 'TcIecLibraryType'}
	{attribute 'external_name' := 'F_VN_InsertIntoContainer_TcVnVector4_INT_GUID_0AC1235C_9EFE_3C53_1027_C594B83B963C'}
	(* Insert an element of type TcVnVector4_INT into a container before the specified position. *)
	FUNCTION F_VN_InsertIntoContainer_TcVnVector4_INT : HRESULT
	VAR_INPUT
		aElement	:	REFERENCE TO TcVnVector4_INT;	(* Single element to insert into ipContainer *)
		ipContainer	:	ITcVnContainer;	(* Container in which to insert the element *)
		nIndex	:	ULINT;	(* Position, before which the element will be inserted *)
		hrPrev	:	HRESULT;	(* HRESULT indicating the result of previous operations (If SUCCEEDED(hrPrev) equals false, no operation is executed.) *)
	END_VAR

END_FUNCTION

// Functions/Basic Container Operations/F_VN_InsertIntoContainer/F_VN_InsertIntoContainer_TcVnVector4_LREAL

	{attribute 'TcIecLibraryType'}
	{attribute 'external_name' := 'F_VN_InsertIntoContainer_TcVnVector4_LREAL_GUID_91F6761F_AF40_3A2B_2782_6CFAA2C6A0F4'}
	(* Insert an element of type TcVnVector4_LREAL into a container before the specified position. *)
	FUNCTION F_VN_InsertIntoContainer_TcVnVector4_LREAL : HRESULT
	VAR_INPUT
		aElement	:	REFERENCE TO TcVnVector4_LREAL;	(* Single element to insert into ipContainer *)
		ipContainer	:	ITcVnContainer;	(* Container in which to insert the element *)
		nIndex	:	ULINT;	(* Position, before which the element will be inserted *)
		hrPrev	:	HRESULT;	(* HRESULT indicating the result of previous operations (If SUCCEEDED(hrPrev) equals false, no operation is executed.) *)
	END_VAR

END_FUNCTION

// Functions/Basic Container Operations/F_VN_InsertIntoContainer/F_VN_InsertIntoContainer_TcVnVector4_SINT

	{attribute 'TcIecLibraryType'}
	{attribute 'external_name' := 'F_VN_InsertIntoContainer_TcVnVector4_SINT_GUID_8A3F9EC8_4594_3F2D_0411_0DD1D850170E'}
	(* Insert an element of type TcVnVector4_SINT into a container before the specified position. *)
	FUNCTION F_VN_InsertIntoContainer_TcVnVector4_SINT : HRESULT
	VAR_INPUT
		aElement	:	REFERENCE TO TcVnVector4_SINT;	(* Single element to insert into ipContainer *)
		ipContainer	:	ITcVnContainer;	(* Container in which to insert the element *)
		nIndex	:	ULINT;	(* Position, before which the element will be inserted *)
		hrPrev	:	HRESULT;	(* HRESULT indicating the result of previous operations (If SUCCEEDED(hrPrev) equals false, no operation is executed.) *)
	END_VAR

END_FUNCTION

// Functions/Basic Container Operations/F_VN_InsertIntoContainer/F_VN_InsertIntoContainer_TcVnVector4_UINT

	{attribute 'TcIecLibraryType'}
	{attribute 'external_name' := 'F_VN_InsertIntoContainer_TcVnVector4_UINT_GUID_3D0DC049_5092_3B34_077D_CE015866C7FE'}
	(* Insert an element of type TcVnVector4_UINT into a container before the specified position. *)
	FUNCTION F_VN_InsertIntoContainer_TcVnVector4_UINT : HRESULT
	VAR_INPUT
		aElement	:	REFERENCE TO TcVnVector4_UINT;	(* Single element to insert into ipContainer *)
		ipContainer	:	ITcVnContainer;	(* Container in which to insert the element *)
		nIndex	:	ULINT;	(* Position, before which the element will be inserted *)
		hrPrev	:	HRESULT;	(* HRESULT indicating the result of previous operations (If SUCCEEDED(hrPrev) equals false, no operation is executed.) *)
	END_VAR

END_FUNCTION

// Functions/Basic Container Operations/F_VN_InsertIntoContainer/F_VN_InsertIntoContainer_TcVnVector4_USINT

	{attribute 'TcIecLibraryType'}
	{attribute 'external_name' := 'F_VN_InsertIntoContainer_TcVnVector4_USINT_GUID_E2B83724_E159_36E5_03EF_04BA02FE2F44'}
	(* Insert an element of type TcVnVector4_USINT into a container before the specified position. *)
	FUNCTION F_VN_InsertIntoContainer_TcVnVector4_USINT : HRESULT
	VAR_INPUT
		aElement	:	REFERENCE TO TcVnVector4_USINT;	(* Single element to insert into ipContainer *)
		ipContainer	:	ITcVnContainer;	(* Container in which to insert the element *)
		nIndex	:	ULINT;	(* Position, before which the element will be inserted *)
		hrPrev	:	HRESULT;	(* HRESULT indicating the result of previous operations (If SUCCEEDED(hrPrev) equals false, no operation is executed.) *)
	END_VAR

END_FUNCTION

// Functions/Basic Container Operations/F_VN_InsertIntoContainer/F_VN_InsertIntoContainer_UDINT

	{attribute 'TcIecLibraryType'}
	{attribute 'external_name' := 'F_VN_InsertIntoContainer_UDINT_GUID_2AC42A46_8B0E_31B9_19A8_34934056B808'}
	(* Insert an element of type UDINT into a container before the specified position. *)
	FUNCTION F_VN_InsertIntoContainer_UDINT : HRESULT
	VAR_INPUT
		nElement	:	UDINT;	(* Single element to insert into ipContainer *)
		ipContainer	:	ITcVnContainer;	(* Container in which to insert the element *)
		nIndex	:	ULINT;	(* Position, before which the element will be inserted *)
		hrPrev	:	HRESULT;	(* HRESULT indicating the result of previous operations (If SUCCEEDED(hrPrev) equals false, no operation is executed.) *)
	END_VAR

END_FUNCTION

// Functions/Basic Container Operations/F_VN_InsertIntoContainer/F_VN_InsertIntoContainer_UINT

	{attribute 'TcIecLibraryType'}
	{attribute 'external_name' := 'F_VN_InsertIntoContainer_UINT_GUID_04E9ECBC_3168_3AE1_1B06_FEB87147868B'}
	(* Insert an element of type UINT into a container before the specified position. *)
	FUNCTION F_VN_InsertIntoContainer_UINT : HRESULT
	VAR_INPUT
		nElement	:	UINT;	(* Single element to insert into ipContainer *)
		ipContainer	:	ITcVnContainer;	(* Container in which to insert the element *)
		nIndex	:	ULINT;	(* Position, before which the element will be inserted *)
		hrPrev	:	HRESULT;	(* HRESULT indicating the result of previous operations (If SUCCEEDED(hrPrev) equals false, no operation is executed.) *)
	END_VAR

END_FUNCTION

// Functions/Basic Container Operations/F_VN_InsertIntoContainer/F_VN_InsertIntoContainer_ULINT

	{attribute 'TcIecLibraryType'}
	{attribute 'external_name' := 'F_VN_InsertIntoContainer_ULINT_GUID_91BD4329_278A_3018_1BB7_637054671FF8'}
	(* Insert an element of type ULINT into a container before the specified position. *)
	FUNCTION F_VN_InsertIntoContainer_ULINT : HRESULT
	VAR_INPUT
		nElement	:	ULINT;	(* Single element to insert into ipContainer *)
		ipContainer	:	ITcVnContainer;	(* Container in which to insert the element *)
		nIndex	:	ULINT;	(* Position, before which the element will be inserted *)
		hrPrev	:	HRESULT;	(* HRESULT indicating the result of previous operations (If SUCCEEDED(hrPrev) equals false, no operation is executed.) *)
	END_VAR

END_FUNCTION

// Functions/Basic Container Operations/F_VN_InsertIntoContainer/F_VN_InsertIntoContainer_USINT

	{attribute 'TcIecLibraryType'}
	{attribute 'external_name' := 'F_VN_InsertIntoContainer_USINT_GUID_C7FF3090_E8BA_3FD7_3A7B_5B3F25D83970'}
	(* Insert an element of type USINT into a container before the specified position. *)
	FUNCTION F_VN_InsertIntoContainer_USINT : HRESULT
	VAR_INPUT
		nElement	:	USINT;	(* Single element to insert into ipContainer *)
		ipContainer	:	ITcVnContainer;	(* Container in which to insert the element *)
		nIndex	:	ULINT;	(* Position, before which the element will be inserted *)
		hrPrev	:	HRESULT;	(* HRESULT indicating the result of previous operations (If SUCCEEDED(hrPrev) equals false, no operation is executed.) *)
	END_VAR

END_FUNCTION

// Functions/Basic Container Operations/F_VN_SetAt/F_VN_SetAt_ITcVnContainer

	{attribute 'TcIecLibraryType'}
	{attribute 'external_name' := 'F_VN_SetAt_ITcVnContainer_GUID_DB775E02_A484_3993_2A91_7F2864122A48'}
	(* Sets the element at the specified index of the container. (Alternatively use interface method .SetAt.) *)
	FUNCTION F_VN_SetAt_ITcVnContainer : HRESULT
	VAR_INPUT
		ipElement	:	ITcVnContainer;	(* Element to set at the specified container position *)
		ipContainer	:	ITcVnContainer;	(* Container with ITcVnContainer elements, in which the element at position nIndex is replaced by ipElement *)
		nIndex	:	ULINT;	(* Index *)
		hrPrev	:	HRESULT;	(* HRESULT indicating the result of previous operations (If SUCCEEDED(hrPrev) equals false, no operation is executed.) *)
	END_VAR

END_FUNCTION

// Functions/Basic Container Operations/F_VN_SetAt/F_VN_SetAt_DINT

	{attribute 'TcIecLibraryType'}
	{attribute 'external_name' := 'F_VN_SetAt_DINT_GUID_4A940B20_8A03_394E_150F_9DA52200395F'}
	(* Sets the element at the specified index of the container. *)
	FUNCTION F_VN_SetAt_DINT : HRESULT
	VAR_INPUT
		nElement	:	DINT;	(* Element to set at the specified container position *)
		ipContainer	:	ITcVnContainer;	(* Container with DINT elements, in which the element at position nIndex is replaced by nElement *)
		nIndex	:	ULINT;	(* Index *)
		hrPrev	:	HRESULT;	(* HRESULT indicating the result of previous operations (If SUCCEEDED(hrPrev) equals false, no operation is executed.) *)
	END_VAR

END_FUNCTION

// Functions/Basic Container Operations/F_VN_SetAt/F_VN_SetAt_INT

	{attribute 'TcIecLibraryType'}
	{attribute 'external_name' := 'F_VN_SetAt_INT_GUID_DF42CE3E_BA33_3691_38B5_EE9DD74CC867'}
	(* Sets the element at the specified index of the container. *)
	FUNCTION F_VN_SetAt_INT : HRESULT
	VAR_INPUT
		nElement	:	INT;	(* Element to set at the specified container position *)
		ipContainer	:	ITcVnContainer;	(* Container with INT elements, in which the element at position nIndex is replaced by nElement *)
		nIndex	:	ULINT;	(* Index *)
		hrPrev	:	HRESULT;	(* HRESULT indicating the result of previous operations (If SUCCEEDED(hrPrev) equals false, no operation is executed.) *)
	END_VAR

END_FUNCTION

// Functions/Basic Container Operations/F_VN_SetAt/F_VN_SetAt_LREAL

	{attribute 'TcIecLibraryType'}
	{attribute 'external_name' := 'F_VN_SetAt_LREAL_GUID_DE239A74_2D13_3DAC_16E1_7EABE24CAE3F'}
	(* Sets the element at the specified index of the container. *)
	FUNCTION F_VN_SetAt_LREAL : HRESULT
	VAR_INPUT
		fElement	:	LREAL;	(* Element to set at the specified container position *)
		ipContainer	:	ITcVnContainer;	(* Container with LREAL elements, in which the element at position nIndex is replaced by fElement *)
		nIndex	:	ULINT;	(* Index *)
		hrPrev	:	HRESULT;	(* HRESULT indicating the result of previous operations (If SUCCEEDED(hrPrev) equals false, no operation is executed.) *)
	END_VAR

END_FUNCTION

// Functions/Basic Container Operations/F_VN_SetAt/F_VN_SetAt_REAL

	{attribute 'TcIecLibraryType'}
	{attribute 'external_name' := 'F_VN_SetAt_REAL_GUID_11354481_31CA_31C2_0398_A02C46E463A3'}
	(* Sets the element at the specified index of the container. *)
	FUNCTION F_VN_SetAt_REAL : HRESULT
	VAR_INPUT
		fElement	:	REAL;	(* Element to set at the specified container position *)
		ipContainer	:	ITcVnContainer;	(* Container with REAL elements, in which the element at position nIndex is replaced by fElement *)
		nIndex	:	ULINT;	(* Index *)
		hrPrev	:	HRESULT;	(* HRESULT indicating the result of previous operations (If SUCCEEDED(hrPrev) equals false, no operation is executed.) *)
	END_VAR

END_FUNCTION

// Functions/Basic Container Operations/F_VN_SetAt/F_VN_SetAt_SINT

	{attribute 'TcIecLibraryType'}
	{attribute 'external_name' := 'F_VN_SetAt_SINT_GUID_CFE9BA93_A5A9_306E_2B7B_3E924AC8D719'}
	(* Sets the element at the specified index of the container. *)
	FUNCTION F_VN_SetAt_SINT : HRESULT
	VAR_INPUT
		nElement	:	SINT;	(* Element to set at the specified container position *)
		ipContainer	:	ITcVnContainer;	(* Container with SINT elements, in which the element at position nIndex is replaced by nElement *)
		nIndex	:	ULINT;	(* Index *)
		hrPrev	:	HRESULT;	(* HRESULT indicating the result of previous operations (If SUCCEEDED(hrPrev) equals false, no operation is executed.) *)
	END_VAR

END_FUNCTION

// Functions/Basic Container Operations/F_VN_SetAt/F_VN_SetAt_TcVnDMatch

	{attribute 'TcIecLibraryType'}
	{attribute 'external_name' := 'F_VN_SetAt_TcVnDMatch_GUID_4276B863_274D_3778_3398_6B8A94BC9E3E'}
	(* Sets the element at the specified index of the container. *)
	FUNCTION F_VN_SetAt_TcVnDMatch : HRESULT
	VAR_INPUT
		stElement	:	REFERENCE TO TcVnDMatch;	(* Element to set at the specified container position *)
		ipContainer	:	ITcVnContainer;	(* Container with TcVnDMatch elements, in which the element at position nIndex is replaced by stElement *)
		nIndex	:	ULINT;	(* Index *)
		hrPrev	:	HRESULT;	(* HRESULT indicating the result of previous operations (If SUCCEEDED(hrPrev) equals false, no operation is executed.) *)
	END_VAR

END_FUNCTION

// Functions/Basic Container Operations/F_VN_SetAt/F_VN_SetAt_TcVnKeyPoint

	{attribute 'TcIecLibraryType'}
	{attribute 'external_name' := 'F_VN_SetAt_TcVnKeyPoint_GUID_3AE28ACB_D61F_3B30_283A_3930209D33A2'}
	(* Sets the element at the specified index of the container. *)
	FUNCTION F_VN_SetAt_TcVnKeyPoint : HRESULT
	VAR_INPUT
		stElement	:	REFERENCE TO TcVnKeyPoint;	(* Element to set at the specified container position *)
		ipContainer	:	ITcVnContainer;	(* Container with TcVnKeyPoint elements, in which the element at position nIndex is replaced by stElement *)
		nIndex	:	ULINT;	(* Index *)
		hrPrev	:	HRESULT;	(* HRESULT indicating the result of previous operations (If SUCCEEDED(hrPrev) equals false, no operation is executed.) *)
	END_VAR

END_FUNCTION

// Functions/Basic Container Operations/F_VN_SetAt/F_VN_SetAt_TcVnPoint2_DINT

	{attribute 'TcIecLibraryType'}
	{attribute 'external_name' := 'F_VN_SetAt_TcVnPoint2_DINT_GUID_57AC02C3_0B1E_37E4_1687_604B77F75A2A'}
	(* Sets the element at the specified index of the container. *)
	FUNCTION F_VN_SetAt_TcVnPoint2_DINT : HRESULT
	VAR_INPUT
		aElement	:	REFERENCE TO TcVnPoint2_DINT;	(* Element to set at the specified container position *)
		ipContainer	:	ITcVnContainer;	(* Container with TcVnPoint2_DINT elements, in which the element at position nIndex is replaced by aElement *)
		nIndex	:	ULINT;	(* Index *)
		hrPrev	:	HRESULT;	(* HRESULT indicating the result of previous operations (If SUCCEEDED(hrPrev) equals false, no operation is executed.) *)
	END_VAR

END_FUNCTION

// Functions/Basic Container Operations/F_VN_SetAt/F_VN_SetAt_TcVnPoint2_LREAL

	{attribute 'TcIecLibraryType'}
	{attribute 'external_name' := 'F_VN_SetAt_TcVnPoint2_LREAL_GUID_5C95F7F6_4DF2_3485_0EFD_DC5D73B7B4E5'}
	(* Sets the element at the specified index of the container. *)
	FUNCTION F_VN_SetAt_TcVnPoint2_LREAL : HRESULT
	VAR_INPUT
		aElement	:	REFERENCE TO TcVnPoint2_LREAL;	(* Element to set at the specified container position *)
		ipContainer	:	ITcVnContainer;	(* Container with TcVnPoint2_LREAL elements, in which the element at position nIndex is replaced by aElement *)
		nIndex	:	ULINT;	(* Index *)
		hrPrev	:	HRESULT;	(* HRESULT indicating the result of previous operations (If SUCCEEDED(hrPrev) equals false, no operation is executed.) *)
	END_VAR

END_FUNCTION

// Functions/Basic Container Operations/F_VN_SetAt/F_VN_SetAt_TcVnPoint2_REAL

	{attribute 'TcIecLibraryType'}
	{attribute 'external_name' := 'F_VN_SetAt_TcVnPoint2_REAL_GUID_0C9C6F68_FF15_38C0_3525_BE44586A7915'}
	(* Sets the element at the specified index of the container. *)
	FUNCTION F_VN_SetAt_TcVnPoint2_REAL : HRESULT
	VAR_INPUT
		aElement	:	REFERENCE TO TcVnPoint2_REAL;	(* Element to set at the specified container position *)
		ipContainer	:	ITcVnContainer;	(* Container with TcVnPoint2_REAL elements, in which the element at position nIndex is replaced by aElement *)
		nIndex	:	ULINT;	(* Index *)
		hrPrev	:	HRESULT;	(* HRESULT indicating the result of previous operations (If SUCCEEDED(hrPrev) equals false, no operation is executed.) *)
	END_VAR

END_FUNCTION

// Functions/Basic Container Operations/F_VN_SetAt/F_VN_SetAt_TcVnPoint3_LREAL

	{attribute 'TcIecLibraryType'}
	{attribute 'external_name' := 'F_VN_SetAt_TcVnPoint3_LREAL_GUID_95A64A79_BA82_35DA_3DB0_8F788CC902F9'}
	(* Sets the element at the specified index of the container. *)
	FUNCTION F_VN_SetAt_TcVnPoint3_LREAL : HRESULT
	VAR_INPUT
		aElement	:	REFERENCE TO TcVnPoint3_LREAL;	(* Element to set at the specified container position *)
		ipContainer	:	ITcVnContainer;	(* Container with TcVnPoint3_LREAL elements, in which the element at position nIndex is replaced by aElement *)
		nIndex	:	ULINT;	(* Index *)
		hrPrev	:	HRESULT;	(* HRESULT indicating the result of previous operations (If SUCCEEDED(hrPrev) equals false, no operation is executed.) *)
	END_VAR

END_FUNCTION

// Functions/Basic Container Operations/F_VN_SetAt/F_VN_SetAt_TcVnPoint3_REAL

	{attribute 'TcIecLibraryType'}
	{attribute 'external_name' := 'F_VN_SetAt_TcVnPoint3_REAL_GUID_A6B321E6_C7C9_3AD9_07B8_40C7F6101D39'}
	(* Sets the element at the specified index of the container. *)
	FUNCTION F_VN_SetAt_TcVnPoint3_REAL : HRESULT
	VAR_INPUT
		aElement	:	REFERENCE TO TcVnPoint3_REAL;	(* Element to set at the specified container position *)
		ipContainer	:	ITcVnContainer;	(* Container with TcVnPoint3_REAL elements, in which the element at position nIndex is replaced by aElement *)
		nIndex	:	ULINT;	(* Index *)
		hrPrev	:	HRESULT;	(* HRESULT indicating the result of previous operations (If SUCCEEDED(hrPrev) equals false, no operation is executed.) *)
	END_VAR

END_FUNCTION

// Functions/Basic Container Operations/F_VN_SetAt/F_VN_SetAt_TcVnRectangle_DINT

	{attribute 'TcIecLibraryType'}
	{attribute 'external_name' := 'F_VN_SetAt_TcVnRectangle_DINT_GUID_2A92903A_445A_3E98_27DB_6DF2DBDF17D8'}
	(* Sets the element at the specified index of the container. *)
	FUNCTION F_VN_SetAt_TcVnRectangle_DINT : HRESULT
	VAR_INPUT
		stElement	:	REFERENCE TO TcVnRectangle_DINT;	(* Element to set at the specified container position *)
		ipContainer	:	ITcVnContainer;	(* Container with TcVnRectangle_DINT elements, in which the element at position nIndex is replaced by stElement *)
		nIndex	:	ULINT;	(* Index *)
		hrPrev	:	HRESULT;	(* HRESULT indicating the result of previous operations (If SUCCEEDED(hrPrev) equals false, no operation is executed.) *)
	END_VAR

END_FUNCTION

// Functions/Basic Container Operations/F_VN_SetAt/F_VN_SetAt_TcVnVector2_DINT

	{attribute 'TcIecLibraryType'}
	{attribute 'external_name' := 'F_VN_SetAt_TcVnVector2_DINT_GUID_413C7576_0C5F_34BC_1801_F750BE9519EF'}
	(* Sets the element at the specified index of the container. *)
	FUNCTION F_VN_SetAt_TcVnVector2_DINT : HRESULT
	VAR_INPUT
		aElement	:	REFERENCE TO TcVnVector2_DINT;	(* Element to set at the specified container position *)
		ipContainer	:	ITcVnContainer;	(* Container with TcVnVector2_DINT elements, in which the element at position nIndex is replaced by aElement *)
		nIndex	:	ULINT;	(* Index *)
		hrPrev	:	HRESULT;	(* HRESULT indicating the result of previous operations (If SUCCEEDED(hrPrev) equals false, no operation is executed.) *)
	END_VAR

END_FUNCTION

// Functions/Basic Container Operations/F_VN_SetAt/F_VN_SetAt_TcVnVector2_INT

	{attribute 'TcIecLibraryType'}
	{attribute 'external_name' := 'F_VN_SetAt_TcVnVector2_INT_GUID_856A18BC_B89C_3687_0577_5918339A416F'}
	(* Sets the element at the specified index of the container. *)
	FUNCTION F_VN_SetAt_TcVnVector2_INT : HRESULT
	VAR_INPUT
		aElement	:	REFERENCE TO TcVnVector2_INT;	(* Element to set at the specified container position *)
		ipContainer	:	ITcVnContainer;	(* Container with TcVnVector2_INT elements, in which the element at position nIndex is replaced by aElement *)
		nIndex	:	ULINT;	(* Index *)
		hrPrev	:	HRESULT;	(* HRESULT indicating the result of previous operations (If SUCCEEDED(hrPrev) equals false, no operation is executed.) *)
	END_VAR

END_FUNCTION

// Functions/Basic Container Operations/F_VN_SetAt/F_VN_SetAt_TcVnVector2_REAL

	{attribute 'TcIecLibraryType'}
	{attribute 'external_name' := 'F_VN_SetAt_TcVnVector2_REAL_GUID_934EC11A_0778_320A_1C2B_28DDE131C688'}
	(* Sets the element at the specified index of the container. *)
	FUNCTION F_VN_SetAt_TcVnVector2_REAL : HRESULT
	VAR_INPUT
		aElement	:	REFERENCE TO TcVnVector2_REAL;	(* Element to set at the specified container position *)
		ipContainer	:	ITcVnContainer;	(* Container with TcVnVector2_REAL elements, in which the element at position nIndex is replaced by aElement *)
		nIndex	:	ULINT;	(* Index *)
		hrPrev	:	HRESULT;	(* HRESULT indicating the result of previous operations (If SUCCEEDED(hrPrev) equals false, no operation is executed.) *)
	END_VAR

END_FUNCTION

// Functions/Basic Container Operations/F_VN_SetAt/F_VN_SetAt_TcVnVector2_SINT

	{attribute 'TcIecLibraryType'}
	{attribute 'external_name' := 'F_VN_SetAt_TcVnVector2_SINT_GUID_5EDC71D5_B54A_3A5D_30CC_E1D567BD0D8C'}
	(* Sets the element at the specified index of the container. *)
	FUNCTION F_VN_SetAt_TcVnVector2_SINT : HRESULT
	VAR_INPUT
		aElement	:	REFERENCE TO TcVnVector2_SINT;	(* Element to set at the specified container position *)
		ipContainer	:	ITcVnContainer;	(* Container with TcVnVector2_SINT elements, in which the element at position nIndex is replaced by aElement *)
		nIndex	:	ULINT;	(* Index *)
		hrPrev	:	HRESULT;	(* HRESULT indicating the result of previous operations (If SUCCEEDED(hrPrev) equals false, no operation is executed.) *)
	END_VAR

END_FUNCTION

// Functions/Basic Container Operations/F_VN_SetAt/F_VN_SetAt_TcVnVector2_UINT

	{attribute 'TcIecLibraryType'}
	{attribute 'external_name' := 'F_VN_SetAt_TcVnVector2_UINT_GUID_3EC043B0_1A45_37D3_15DE_3263AC44312B'}
	(* Sets the element at the specified index of the container. *)
	FUNCTION F_VN_SetAt_TcVnVector2_UINT : HRESULT
	VAR_INPUT
		aElement	:	REFERENCE TO TcVnVector2_UINT;	(* Element to set at the specified container position *)
		ipContainer	:	ITcVnContainer;	(* Container with TcVnVector2_UINT elements, in which the element at position nIndex is replaced by aElement *)
		nIndex	:	ULINT;	(* Index *)
		hrPrev	:	HRESULT;	(* HRESULT indicating the result of previous operations (If SUCCEEDED(hrPrev) equals false, no operation is executed.) *)
	END_VAR

END_FUNCTION

// Functions/Basic Container Operations/F_VN_SetAt/F_VN_SetAt_TcVnVector2_USINT

	{attribute 'TcIecLibraryType'}
	{attribute 'external_name' := 'F_VN_SetAt_TcVnVector2_USINT_GUID_6E59FD45_4A72_346E_0E13_03F360DD3B96'}
	(* Sets the element at the specified index of the container. *)
	FUNCTION F_VN_SetAt_TcVnVector2_USINT : HRESULT
	VAR_INPUT
		aElement	:	REFERENCE TO TcVnVector2_USINT;	(* Element to set at the specified container position *)
		ipContainer	:	ITcVnContainer;	(* Container with TcVnVector2_USINT elements, in which the element at position nIndex is replaced by aElement *)
		nIndex	:	ULINT;	(* Index *)
		hrPrev	:	HRESULT;	(* HRESULT indicating the result of previous operations (If SUCCEEDED(hrPrev) equals false, no operation is executed.) *)
	END_VAR

END_FUNCTION

// Functions/Basic Container Operations/F_VN_SetAt/F_VN_SetAt_TcVnVector3_INT

	{attribute 'TcIecLibraryType'}
	{attribute 'external_name' := 'F_VN_SetAt_TcVnVector3_INT_GUID_ACB92D18_4D64_335A_3AF5_197AB7367C34'}
	(* Sets the element at the specified index of the container. *)
	FUNCTION F_VN_SetAt_TcVnVector3_INT : HRESULT
	VAR_INPUT
		aElement	:	REFERENCE TO TcVnVector3_INT;	(* Element to set at the specified container position *)
		ipContainer	:	ITcVnContainer;	(* Container with TcVnVector3_INT elements, in which the element at position nIndex is replaced by aElement *)
		nIndex	:	ULINT;	(* Index *)
		hrPrev	:	HRESULT;	(* HRESULT indicating the result of previous operations (If SUCCEEDED(hrPrev) equals false, no operation is executed.) *)
	END_VAR

END_FUNCTION

// Functions/Basic Container Operations/F_VN_SetAt/F_VN_SetAt_TcVnVector3_REAL

